   1:  PR[GP1:91,2] = PR[GP1:90,2] + -23.131;
   1:L PR[91] 10mm/sec CNT100;
   1:  PR[GP1:91,1] = PR[GP1:90,1] + -1.490;
   1:  PR[GP1:91,2] = PR[GP1:90,2] + -22.735;
   1:L PR[91] 10mm/sec CNT100;
   1:  PR[GP1:91,1] = PR[GP1:90,1] + 0.863;
   1:  PR[GP1:91,2] = PR[GP1:90,2] + -21.488;
   1:L PR[91] 10mm/sec CNT100;
   1:  PR[GP1:91,1] = PR[GP1:90,1] + 4.214;
   1:  PR[GP1:91,2] = PR[GP1:90,2] + -23.194;
   1:L PR[91] 10mm/sec CNT100;
   1:  PR[GP1:91,1] = PR[GP1:90,1] + 6.727;
   1:  PR[GP1:91,2] = PR[GP1:90,2] + -26.111;
   1:L PR[91] 10mm/sec CNT100;
   1:  PR[GP1:91,1] = PR[GP1:90,1] + 10.077;
   1:  PR[GP1:91,2] = PR[GP1:90,2] + -28.732;
   1:L PR[91] 10mm/sec CNT100;
   1:  PR[GP1:91,1] = PR[GP1:90,1] + 11.446;
   1:  PR[GP1:91,2] = PR[GP1:90,2] + -29.727;
   1:L PR[91] 10mm/sec CNT100;
   1:  PR[GP1:91,1] = PR[GP1:90,1] + 16.570;
   1:  PR[GP1:91,2] = PR[GP1:90,2] + -32.401;
   1:L PR[91] 10mm/sec CNT100;
   1:  PR[GP1:91,1] = PR[GP1:90,1] + 22.895;
   1:  PR[GP1:91,2] = PR[GP1:90,2] + -34.433;
   1:L PR[91] 10mm/sec CNT100;
   1:  PR[GP1:91,1] = PR[GP1:90,1] + 23.903;
   1:  PR[GP1:91,2] = PR[GP1:90,2] + -34.782;
   1:L PR[91] 10mm/sec CNT100;
   1:  PR[GP1:91,1] = PR[GP1:90,1] + 30.511;
   1:  PR[GP1:91,2] = PR[GP1:90,2] + -35.650;
   1:L PR[91] 10mm/sec CNT100;
   1:  PR[GP1:91,1] = PR[GP1:90,1] + 37.251;
   1:  PR[GP1:91,2] = PR[GP1:90,2] + -35.453;
   1:L PR[91] 10mm/sec CNT100;
   1:  PR[GP1:91,1] = PR[GP1:90,1] + 39.091;
   1:  PR[GP1:91,2] = PR[GP1:90,2] + -35.024;
   1:L PR[91] 10mm/sec CNT100;
   1:  PR[GP1:91,1] = PR[GP1:90,1] + 45.087;
   1:  PR[GP1:91,2] = PR[GP1:90,2] + -33.728;
   1:L PR[91] 10mm/sec CNT100;
   1:  PR[GP1:91,1] = PR[GP1:90,1] + 48.963;
   1:  PR[GP1:91,2] = PR[GP1:90,2] + -32.210;
   1:L PR[91] 10mm/sec CNT100;
   1:  PR[GP1:91,1] = PR[GP1:90,1] + 53.686;
   1:  PR[GP1:91,2] = PR[GP1:90,2] + -29.527;
   1:L PR[91] 10mm/sec CNT100;
   1:  PR[GP1:91,1] = PR[GP1:90,1] + 56.440;
   1:  PR[GP1:91,2] = PR[GP1:90,2] + -27.829;
   1:L PR[91] 10mm/sec CNT100;
   1:  PR[GP1:91,1] = PR[GP1:90,1] + 58.226;
   1:  PR[GP1:91,2] = PR[GP1:90,2] + -26.233;
   1:L PR[91] 10mm/sec CNT100;
   1:  PR[GP1:91,1] = PR[GP1:90,1] + 63.305;
   1:  PR[GP1:91,2] = PR[GP1:90,2] + -20.876;
   1:L PR[91] 10mm/sec CNT100;
   1:  PR[GP1:91,1] = PR[GP1:90,1] + 64.349;
   1:  PR[GP1:91,2] = PR[GP1:90,2] + -19.525;
   1:L PR[91] 10mm/sec CNT100;
   1:  PR[GP1:91,1] = PR[GP1:90,1] + 68.774;
   1:  PR[GP1:91,2] = PR[GP1:90,2] + -10.736;
   1:L PR[91] 10mm/sec CNT100;
   1:  PR[GP1:91,1] = PR[GP1:90,1] + 69.043;
   1:  PR[GP1:91,2] = PR[GP1:90,2] + -9.836;
   1:L PR[91] 10mm/sec CNT100;
   1:  PR[GP1:91,1] = PR[GP1:90,1] + 70.464;
   1:  PR[GP1:91,2] = PR[GP1:90,2] + -0.697;
   1:L PR[91] 10mm/sec CNT100;
   1:  PR[GP1:91,1] = PR[GP1:90,1] + 70.526;
   1:  PR[GP1:91,2] = PR[GP1:90,2] + -0.024;
   1:L PR[91] 10mm/sec CNT100;
   1:  PR[GP1:91,1] = PR[GP1:90,1] + 69.127;
   1:  PR[GP1:91,2] = PR[GP1:90,2] + 8.859;
   1:L PR[91] 10mm/sec CNT100;
   1:  PR[GP1:91,1] = PR[GP1:90,1] + 69.037;
   1:  PR[GP1:91,2] = PR[GP1:90,2] + 9.845;
   1:L PR[91] 10mm/sec CNT100;
   1:  PR[GP1:91,1] = PR[GP1:90,1] + 68.774;
   1:  PR[GP1:91,2] = PR[GP1:90,2] + 10.728;
   1:L PR[91] 10mm/sec CNT100;
   1:  PR[GP1:91,1] = PR[GP1:90,1] + 64.349;
   1:  PR[GP1:91,2] = PR[GP1:90,2] + 19.516;
   1:L PR[91] 10mm/sec CNT100;
   1:  PR[GP1:91,1] = PR[GP1:90,1] + 63.305;
   1:  PR[GP1:91,2] = PR[GP1:90,2] + 20.868;
   1:L PR[91] 10mm/sec CNT100;
   1:  PR[GP1:91,1] = PR[GP1:90,1] + 58.226;
   1:  PR[GP1:91,2] = PR[GP1:90,2] + 26.224;
   1:L PR[91] 10mm/sec CNT100;
   1:  PR[GP1:91,1] = PR[GP1:90,1] + 56.449;
   1:  PR[GP1:91,2] = PR[GP1:90,2] + 27.812;
   1:L PR[91] 10mm/sec CNT100;
   1:  PR[GP1:91,1] = PR[GP1:90,1] + 51.595;
   1:  PR[GP1:91,2] = PR[GP1:90,2] + 30.539;
   1:L PR[91] 10mm/sec CNT100;
   1:  PR[GP1:91,1] = PR[GP1:90,1] + 48.950;
   1:  PR[GP1:91,2] = PR[GP1:90,2] + 32.206;
   1:L PR[91] 10mm/sec CNT100;
   1:  PR[GP1:91,1] = PR[GP1:90,1] + 45.081;
   1:  PR[GP1:91,2] = PR[GP1:90,2] + 33.721;
   1:L PR[91] 10mm/sec CNT100;
   1:  PR[GP1:91,1] = PR[GP1:90,1] + 41.998;
   1:  PR[GP1:91,2] = PR[GP1:90,2] + 34.448;
   1:L PR[91] 10mm/sec CNT100;
   1:  PR[GP1:91,1] = PR[GP1:90,1] + 37.257;
   1:  PR[GP1:91,2] = PR[GP1:90,2] + 35.444;
   1:L PR[91] 10mm/sec CNT100;
   1:  PR[GP1:91,1] = PR[GP1:90,1] + 30.511;
   1:  PR[GP1:91,2] = PR[GP1:90,2] + 35.642;
   1:L PR[91] 10mm/sec CNT100;
   1:  PR[GP1:91,1] = PR[GP1:90,1] + 23.897;
   1:  PR[GP1:91,2] = PR[GP1:90,2] + 34.772;
   1:L PR[91] 10mm/sec CNT100;
   1:  PR[GP1:91,1] = PR[GP1:90,1] + 18.223;
   1:  PR[GP1:91,2] = PR[GP1:90,2] + 32.967;
   1:L PR[91] 10mm/sec CNT100;
   1:  PR[GP1:91,1] = PR[GP1:90,1] + 16.579;
   1:  PR[GP1:91,2] = PR[GP1:90,2] + 32.397;
   1:L PR[91] 10mm/sec CNT100;
   1:  PR[GP1:91,1] = PR[GP1:90,1] + 11.445;
   1:  PR[GP1:91,2] = PR[GP1:90,2] + 29.717;
   1:L PR[91] 10mm/sec CNT100;
   1:  PR[GP1:91,1] = PR[GP1:90,1] + 10.460;
   1:  PR[GP1:91,2] = PR[GP1:90,2] + 29.022;
   1:L PR[91] 10mm/sec CNT100;
   1:  PR[GP1:91,1] = PR[GP1:90,1] + 6.917;
   1:  PR[GP1:91,2] = PR[GP1:90,2] + 26.249;
   1:L PR[91] 10mm/sec CNT100;
   1:  PR[GP1:91,1] = PR[GP1:90,1] + 4.197;
   1:  PR[GP1:91,2] = PR[GP1:90,2] + 23.083;
   1:L PR[91] 10mm/sec CNT100;
   1:  PR[GP1:91,1] = PR[GP1:90,1] + 3.346;
   1:  PR[GP1:91,2] = PR[GP1:90,2] + 22.747;
   1:L PR[91] 10mm/sec CNT100;
   1:  PR[GP1:91,1] = PR[GP1:90,1] + 0.976;
   1:  PR[GP1:91,2] = PR[GP1:90,2] + 21.536;
   1:L PR[91] 10mm/sec CNT100;
   1:  PR[GP1:91,1] = PR[GP1:90,1] + -0.928;
   1:  PR[GP1:91,2] = PR[GP1:90,2] + 22.512;
   1:  PR[GP1:91,3] = PR[GP1:90,3] + 46.550;
   1:L PR[91] 10mm/sec CNT100;
   1:  PR[GP1:91,1] = PR[GP1:90,1] + -3.325;
   1:  PR[GP1:91,2] = PR[GP1:90,2] + 23.731;
   1:L PR[91] 10mm/sec CNT100;
   1:  PR[GP1:91,1] = PR[GP1:90,1] + -5.725;
   1:  PR[GP1:91,2] = PR[GP1:90,2] + 26.522;
   1:L PR[91] 10mm/sec CNT100;
   1:  PR[GP1:91,1] = PR[GP1:90,1] + -8.906;
   1:  PR[GP1:91,2] = PR[GP1:90,2] + 29.013;
   1:L PR[91] 10mm/sec CNT100;
   1:  PR[GP1:91,1] = PR[GP1:90,1] + -10.149;
   1:  PR[GP1:91,2] = PR[GP1:90,2] + 29.891;
   1:L PR[91] 10mm/sec CNT100;
   1:  PR[GP1:91,1] = PR[GP1:90,1] + -15.022;
   1:  PR[GP1:91,2] = PR[GP1:90,2] + 32.441;
   1:L PR[91] 10mm/sec CNT100;
   1:  PR[GP1:91,1] = PR[GP1:90,1] + -20.991;
   1:  PR[GP1:91,2] = PR[GP1:90,2] + 34.359;
   1:L PR[91] 10mm/sec CNT100;
   1:  PR[GP1:91,1] = PR[GP1:90,1] + -22.656;
   1:  PR[GP1:91,2] = PR[GP1:90,2] + 34.934;
   1:L PR[91] 10mm/sec CNT100;
   1:  PR[GP1:91,1] = PR[GP1:90,1] + -28.937;
   1:  PR[GP1:91,2] = PR[GP1:90,2] + 35.755;
   1:L PR[91] 10mm/sec CNT100;
   1:  PR[GP1:91,1] = PR[GP1:90,1] + -36.208;
   1:  PR[GP1:91,2] = PR[GP1:90,2] + 35.505;
   1:L PR[91] 10mm/sec CNT100;
   1:  PR[GP1:91,1] = PR[GP1:90,1] + -43.441;
   1:  PR[GP1:91,2] = PR[GP1:90,2] + 33.938;
   1:L PR[91] 10mm/sec CNT100;
   1:  PR[GP1:91,1] = PR[GP1:90,1] + -48.169;
   1:  PR[GP1:91,2] = PR[GP1:90,2] + 32.077;
   1:L PR[91] 10mm/sec CNT100;
   1:  PR[GP1:91,1] = PR[GP1:90,1] + -51.524;
   1:  PR[GP1:91,2] = PR[GP1:90,2] + 30.168;
   1:L PR[91] 10mm/sec CNT100;
   1:  PR[GP1:91,1] = PR[GP1:90,1] + -55.181;
   1:  PR[GP1:91,2] = PR[GP1:90,2] + 27.903;
   1:L PR[91] 10mm/sec CNT100;
   1:  PR[GP1:91,1] = PR[GP1:90,1] + -57.555;
   1:  PR[GP1:91,2] = PR[GP1:90,2] + 25.775;
   1:L PR[91] 10mm/sec CNT100;
   1:  PR[GP1:91,1] = PR[GP1:90,1] + -61.710;
   1:  PR[GP1:91,2] = PR[GP1:90,2] + 21.407;
   1:L PR[91] 10mm/sec CNT100;
   1:  PR[GP1:91,1] = PR[GP1:90,1] + -63.266;
   1:  PR[GP1:91,2] = PR[GP1:90,2] + 19.387;
   1:L PR[91] 10mm/sec CNT100;
   1:  PR[GP1:91,1] = PR[GP1:90,1] + -67.485;
   1:  PR[GP1:91,2] = PR[GP1:90,2] + 10.965;
   1:L PR[91] 10mm/sec CNT100;
   1:  PR[GP1:91,1] = PR[GP1:90,1] + -67.973;
   1:  PR[GP1:91,2] = PR[GP1:90,2] + 9.309;
   1:L PR[91] 10mm/sec CNT100;
   1:  PR[GP1:91,1] = PR[GP1:90,1] + -69.196;
   1:  PR[GP1:91,2] = PR[GP1:90,2] + 1.460;
   1:L PR[91] 10mm/sec CNT100;
   1:  PR[GP1:91,1] = PR[GP1:90,1] + -69.326;
   1:  PR[GP1:91,2] = PR[GP1:90,2] + 0.016;
   1:L PR[91] 10mm/sec CNT100;
   1:  PR[GP1:91,1] = PR[GP1:90,1] + -68.117;
   1:  PR[GP1:91,2] = PR[GP1:90,2] + -7.637;
   1:L PR[91] 10mm/sec CNT100;
   1:  PR[GP1:91,1] = PR[GP1:90,1] + -67.967;
   1:  PR[GP1:91,2] = PR[GP1:90,2] + -9.337;
   1:L PR[91] 10mm/sec CNT100;
   1:  PR[GP1:91,1] = PR[GP1:90,1] + -67.485;
   1:  PR[GP1:91,2] = PR[GP1:90,2] + -10.974;
   1:L PR[91] 10mm/sec CNT100;
   1:  PR[GP1:91,1] = PR[GP1:90,1] + -63.266;
   1:  PR[GP1:91,2] = PR[GP1:90,2] + -19.396;
   1:L PR[91] 10mm/sec CNT100;
   1:  PR[GP1:91,1] = PR[GP1:90,1] + -61.710;
   1:  PR[GP1:91,2] = PR[GP1:90,2] + -21.416;
   1:L PR[91] 10mm/sec CNT100;
   1:  PR[GP1:91,1] = PR[GP1:90,1] + -57.555;
   1:  PR[GP1:91,2] = PR[GP1:90,2] + -25.784;
   1:L PR[91] 10mm/sec CNT100;
   1:  PR[GP1:91,1] = PR[GP1:90,1] + -55.191;
   1:  PR[GP1:91,2] = PR[GP1:90,2] + -27.903;
   1:L PR[91] 10mm/sec CNT100;
   1:  PR[GP1:91,1] = PR[GP1:90,1] + -51.401;
   1:  PR[GP1:91,2] = PR[GP1:90,2] + -30.035;
   1:L PR[91] 10mm/sec CNT100;
   1:  PR[GP1:91,1] = PR[GP1:90,1] + -48.156;
   1:  PR[GP1:91,2] = PR[GP1:90,2] + -32.091;
   1:L PR[91] 10mm/sec CNT100;
   1:  PR[GP1:91,1] = PR[GP1:90,1] + -43.436;
   1:  PR[GP1:91,2] = PR[GP1:90,2] + -33.949;
   1:L PR[91] 10mm/sec CNT100;
   1:  PR[GP1:91,1] = PR[GP1:90,1] + -41.730;
   1:  PR[GP1:91,2] = PR[GP1:90,2] + -34.350;
   1:L PR[91] 10mm/sec CNT100;
   1:  PR[GP1:91,1] = PR[GP1:90,1] + -36.208;
   1:  PR[GP1:91,2] = PR[GP1:90,2] + -35.514;
   1:L PR[91] 10mm/sec CNT100;
   1:  PR[GP1:91,1] = PR[GP1:90,1] + -29.774;
   1:  PR[GP1:91,2] = PR[GP1:90,2] + -35.762;
   1:L PR[91] 10mm/sec CNT100;
   1:  PR[GP1:91,1] = PR[GP1:90,1] + -28.945;
   1:  PR[GP1:91,2] = PR[GP1:90,2] + -35.765;
   1:L PR[91] 10mm/sec CNT100;
   1:  PR[GP1:91,1] = PR[GP1:90,1] + -22.646;
   1:  PR[GP1:91,2] = PR[GP1:90,2] + -34.942;
   1:L PR[91] 10mm/sec CNT100;
   1:  PR[GP1:91,1] = PR[GP1:90,1] + -17.264;
   1:  PR[GP1:91,2] = PR[GP1:90,2] + -33.229;
   1:L PR[91] 10mm/sec CNT100;
   1:  PR[GP1:91,1] = PR[GP1:90,1] + -15.025;
   1:  PR[GP1:91,2] = PR[GP1:90,2] + -32.451;
   1:L PR[91] 10mm/sec CNT100;
   1:  PR[GP1:91,1] = PR[GP1:90,1] + -10.150;
   1:  PR[GP1:91,2] = PR[GP1:90,2] + -29.900;
   1:L PR[91] 10mm/sec CNT100;
   1:  PR[GP1:91,1] = PR[GP1:90,1] + -8.426;
   1:  PR[GP1:91,2] = PR[GP1:90,2] + -28.648;
   1:L PR[91] 10mm/sec CNT100;
   1:  PR[GP1:91,1] = PR[GP1:90,1] + -5.499;
   1:  PR[GP1:91,2] = PR[GP1:90,2] + -26.355;
   1:L PR[91] 10mm/sec CNT100;
   1:  PR[GP1:91,1] = PR[GP1:90,1] + -3.269;
   1:  PR[GP1:91,2] = PR[GP1:90,2] + -23.769;
   1:L PR[91] 10mm/sec CNT100;
   1:  PR[GP1:91,1] = PR[GP1:90,1] + -1.127;
   1:  PR[GP1:91,2] = PR[GP1:90,2] + -23.309;
   1:L PR[91] 10mm/sec CNT100;
   1:  PR[GP1:91,1] = PR[GP1:90,1] + 0.953;
   1:  PR[GP1:91,2] = PR[GP1:90,2] + -22.208;
   1:L PR[91] 10mm/sec CNT100;
   1:  PR[GP1:91,1] = PR[GP1:90,1] + 4.149;
   1:  PR[GP1:91,2] = PR[GP1:90,2] + -23.833;
   1:L PR[91] 10mm/sec CNT100;
   1:  PR[GP1:91,1] = PR[GP1:90,1] + 6.345;
   1:  PR[GP1:91,2] = PR[GP1:90,2] + -26.382;
   1:L PR[91] 10mm/sec CNT100;
   1:  PR[GP1:91,1] = PR[GP1:90,1] + 9.258;
   1:  PR[GP1:91,2] = PR[GP1:90,2] + -28.661;
   1:L PR[91] 10mm/sec CNT100;
   1:  PR[GP1:91,1] = PR[GP1:90,1] + 10.985;
   1:  PR[GP1:91,2] = PR[GP1:90,2] + -29.916;
   1:L PR[91] 10mm/sec CNT100;
   1:  PR[GP1:91,1] = PR[GP1:90,1] + 15.824;
   1:  PR[GP1:91,2] = PR[GP1:90,2] + -32.441;
   1:L PR[91] 10mm/sec CNT100;
   1:  PR[GP1:91,1] = PR[GP1:90,1] + 21.801;
   1:  PR[GP1:91,2] = PR[GP1:90,2] + -34.362;
   1:L PR[91] 10mm/sec CNT100;
   1:  PR[GP1:91,1] = PR[GP1:90,1] + 23.469;
   1:  PR[GP1:91,2] = PR[GP1:90,2] + -34.939;
   1:L PR[91] 10mm/sec CNT100;
   1:  PR[GP1:91,1] = PR[GP1:90,1] + 29.742;
   1:  PR[GP1:91,2] = PR[GP1:90,2] + -35.764;
   1:L PR[91] 10mm/sec CNT100;
   1:  PR[GP1:91,1] = PR[GP1:90,1] + 36.985;
   1:  PR[GP1:91,2] = PR[GP1:90,2] + -35.521;
   1:L PR[91] 10mm/sec CNT100;
   1:  PR[GP1:91,1] = PR[GP1:90,1] + 44.219;
   1:  PR[GP1:91,2] = PR[GP1:90,2] + -33.956;
   1:L PR[91] 10mm/sec CNT100;
   1:  PR[GP1:91,1] = PR[GP1:90,1] + 48.968;
   1:  PR[GP1:91,2] = PR[GP1:90,2] + -32.097;
   1:L PR[91] 10mm/sec CNT100;
   1:  PR[GP1:91,1] = PR[GP1:90,1] + 52.319;
   1:  PR[GP1:91,2] = PR[GP1:90,2] + -30.193;
   1:L PR[91] 10mm/sec CNT100;
   1:  PR[GP1:91,1] = PR[GP1:90,1] + 55.967;
   1:  PR[GP1:91,2] = PR[GP1:90,2] + -27.944;
   1:L PR[91] 10mm/sec CNT100;
   1:  PR[GP1:91,1] = PR[GP1:90,1] + 58.339;
   1:  PR[GP1:91,2] = PR[GP1:90,2] + -25.825;
   1:L PR[91] 10mm/sec CNT100;
   1:  PR[GP1:91,1] = PR[GP1:90,1] + 62.493;
   1:  PR[GP1:91,2] = PR[GP1:90,2] + -21.443;
   1:L PR[91] 10mm/sec CNT100;
   1:  PR[GP1:91,1] = PR[GP1:90,1] + 64.073;
   1:  PR[GP1:91,2] = PR[GP1:90,2] + -19.399;
   1:L PR[91] 10mm/sec CNT100;
   1:  PR[GP1:91,1] = PR[GP1:90,1] + 67.337;
   1:  PR[GP1:91,2] = PR[GP1:90,2] + -12.902;
   1:L PR[91] 10mm/sec CNT100;
   1:  PR[GP1:91,1] = PR[GP1:90,1] + 68.299;
   1:  PR[GP1:91,2] = PR[GP1:90,2] + -11.018;
   1:L PR[91] 10mm/sec CNT100;
   1:  PR[GP1:91,1] = PR[GP1:90,1] + 68.786;
   1:  PR[GP1:91,2] = PR[GP1:90,2] + -9.386;
   1:L PR[91] 10mm/sec CNT100;
   1:  PR[GP1:91,1] = PR[GP1:90,1] + 70.010;
   1:  PR[GP1:91,2] = PR[GP1:90,2] + -1.512;
   1:L PR[91] 10mm/sec CNT100;
   1:  PR[GP1:91,1] = PR[GP1:90,1] + 70.147;
   1:  PR[GP1:91,2] = PR[GP1:90,2] + -0.024;
   1:L PR[91] 10mm/sec CNT100;
   1:  PR[GP1:91,1] = PR[GP1:90,1] + 68.938;
   1:  PR[GP1:91,2] = PR[GP1:90,2] + 7.649;
   1:L PR[91] 10mm/sec CNT100;
   1:  PR[GP1:91,1] = PR[GP1:90,1] + 68.780;
   1:  PR[GP1:91,2] = PR[GP1:90,2] + 9.396;
   1:L PR[91] 10mm/sec CNT100;
   1:  PR[GP1:91,1] = PR[GP1:90,1] + 68.298;
   1:  PR[GP1:91,2] = PR[GP1:90,2] + 11.011;
   1:L PR[91] 10mm/sec CNT100;
   1:  PR[GP1:91,1] = PR[GP1:90,1] + 65.100;
   1:  PR[GP1:91,2] = PR[GP1:90,2] + 17.382;
   1:L PR[91] 10mm/sec CNT100;
   1:  PR[GP1:91,1] = PR[GP1:90,1] + 64.074;
   1:  PR[GP1:91,2] = PR[GP1:90,2] + 19.388;
   1:L PR[91] 10mm/sec CNT100;
   1:  PR[GP1:91,1] = PR[GP1:90,1] + 62.493;
   1:  PR[GP1:91,2] = PR[GP1:90,2] + 21.434;
   1:L PR[91] 10mm/sec CNT100;
   1:  PR[GP1:91,1] = PR[GP1:90,1] + 58.339;
   1:  PR[GP1:91,2] = PR[GP1:90,2] + 25.816;
   1:L PR[91] 10mm/sec CNT100;
   1:  PR[GP1:91,1] = PR[GP1:90,1] + 55.976;
   1:  PR[GP1:91,2] = PR[GP1:90,2] + 27.927;
   1:L PR[91] 10mm/sec CNT100;
   1:  PR[GP1:91,1] = PR[GP1:90,1] + 52.190;
   1:  PR[GP1:91,2] = PR[GP1:90,2] + 30.054;
   1:L PR[91] 10mm/sec CNT100;
   1:  PR[GP1:91,1] = PR[GP1:90,1] + 48.955;
   1:  PR[GP1:91,2] = PR[GP1:90,2] + 32.093;
   1:L PR[91] 10mm/sec CNT100;
   1:  PR[GP1:91,1] = PR[GP1:90,1] + 44.214;
   1:  PR[GP1:91,2] = PR[GP1:90,2] + 33.949;
   1:L PR[91] 10mm/sec CNT100;
   1:  PR[GP1:91,1] = PR[GP1:90,1] + 42.517;
   1:  PR[GP1:91,2] = PR[GP1:90,2] + 34.349;
   1:L PR[91] 10mm/sec CNT100;
   1:  PR[GP1:91,1] = PR[GP1:90,1] + 36.985;
   1:  PR[GP1:91,2] = PR[GP1:90,2] + 35.512;
   1:L PR[91] 10mm/sec CNT100;
   1:  PR[GP1:91,1] = PR[GP1:90,1] + 30.583;
   1:  PR[GP1:91,2] = PR[GP1:90,2] + 35.753;
   1:L PR[91] 10mm/sec CNT100;
   1:  PR[GP1:91,1] = PR[GP1:90,1] + 29.753;
   1:  PR[GP1:91,2] = PR[GP1:90,2] + 35.756;
   1:L PR[91] 10mm/sec CNT100;
   1:  PR[GP1:91,1] = PR[GP1:90,1] + 23.464;
   1:  PR[GP1:91,2] = PR[GP1:90,2] + 34.930;
   1:L PR[91] 10mm/sec CNT100;
   1:  PR[GP1:91,1] = PR[GP1:90,1] + 18.075;
   1:  PR[GP1:91,2] = PR[GP1:90,2] + 33.215;
   1:L PR[91] 10mm/sec CNT100;
   1:  PR[GP1:91,1] = PR[GP1:90,1] + 15.834;
   1:  PR[GP1:91,2] = PR[GP1:90,2] + 32.438;
   1:L PR[91] 10mm/sec CNT100;
   1:  PR[GP1:91,1] = PR[GP1:90,1] + 10.984;
   1:  PR[GP1:91,2] = PR[GP1:90,2] + 29.907;
   1:L PR[91] 10mm/sec CNT100;
   1:  PR[GP1:91,1] = PR[GP1:90,1] + 9.739;
   1:  PR[GP1:91,2] = PR[GP1:90,2] + 29.027;
   1:L PR[91] 10mm/sec CNT100;
   1:  PR[GP1:91,1] = PR[GP1:90,1] + 6.573;
   1:  PR[GP1:91,2] = PR[GP1:90,2] + 26.550;
   1:L PR[91] 10mm/sec CNT100;
   1:  PR[GP1:91,1] = PR[GP1:90,1] + 4.132;
   1:  PR[GP1:91,2] = PR[GP1:90,2] + 23.708;
   1:L PR[91] 10mm/sec CNT100;
   1:  PR[GP1:91,1] = PR[GP1:90,1] + 3.152;
   1:  PR[GP1:91,2] = PR[GP1:90,2] + 23.322;
   1:L PR[91] 10mm/sec CNT100;
   1:  PR[GP1:91,1] = PR[GP1:90,1] + 1.066;
   1:  PR[GP1:91,2] = PR[GP1:90,2] + 22.256;
   1:L PR[91] 10mm/sec CNT100;
   1:  PR[GP1:91,1] = PR[GP1:90,1] + -1.121;
   1:  PR[GP1:91,2] = PR[GP1:90,2] + 23.268;
   1:  PR[GP1:91,3] = PR[GP1:90,3] + 47.880;
   1:L PR[91] 10mm/sec CNT100;
   1:  PR[GP1:91,1] = PR[GP1:90,1] + -3.261;
   1:  PR[GP1:91,2] = PR[GP1:90,2] + 24.356;
   1:L PR[91] 10mm/sec CNT100;
   1:  PR[GP1:91,1] = PR[GP1:90,1] + -5.385;
   1:  PR[GP1:91,2] = PR[GP1:90,2] + 26.826;
   1:L PR[91] 10mm/sec CNT100;
   1:  PR[GP1:91,1] = PR[GP1:90,1] + -8.188;
   1:  PR[GP1:91,2] = PR[GP1:90,2] + 29.021;
   1:L PR[91] 10mm/sec CNT100;
   1:  PR[GP1:91,1] = PR[GP1:90,1] + -9.689;
   1:  PR[GP1:91,2] = PR[GP1:90,2] + 30.082;
   1:L PR[91] 10mm/sec CNT100;
   1:  PR[GP1:91,1] = PR[GP1:90,1] + -14.277;
   1:  PR[GP1:91,2] = PR[GP1:90,2] + 32.482;
   1:L PR[91] 10mm/sec CNT100;
   1:  PR[GP1:91,1] = PR[GP1:90,1] + -19.899;
   1:  PR[GP1:91,2] = PR[GP1:90,2] + 34.288;
   1:L PR[91] 10mm/sec CNT100;
   1:  PR[GP1:91,1] = PR[GP1:90,1] + -22.224;
   1:  PR[GP1:91,2] = PR[GP1:90,2] + 35.092;
   1:L PR[91] 10mm/sec CNT100;
   1:  PR[GP1:91,1] = PR[GP1:90,1] + -28.171;
   1:  PR[GP1:91,2] = PR[GP1:90,2] + 35.869;
   1:L PR[91] 10mm/sec CNT100;
   1:  PR[GP1:91,1] = PR[GP1:90,1] + -35.111;
   1:  PR[GP1:91,2] = PR[GP1:90,2] + 35.630;
   1:L PR[91] 10mm/sec CNT100;
   1:  PR[GP1:91,1] = PR[GP1:90,1] + -35.807;
   1:  PR[GP1:91,2] = PR[GP1:90,2] + 35.627;
   1:L PR[91] 10mm/sec CNT100;
   1:  PR[GP1:91,1] = PR[GP1:90,1] + -42.581;
   1:  PR[GP1:91,2] = PR[GP1:90,2] + 34.164;
   1:L PR[91] 10mm/sec CNT100;
   1:  PR[GP1:91,1] = PR[GP1:90,1] + -48.178;
   1:  PR[GP1:91,2] = PR[GP1:90,2] + 31.961;
   1:L PR[91] 10mm/sec CNT100;
   1:  PR[GP1:91,1] = PR[GP1:90,1] + -50.163;
   1:  PR[GP1:91,2] = PR[GP1:90,2] + 30.832;
   1:L PR[91] 10mm/sec CNT100;
   1:  PR[GP1:91,1] = PR[GP1:90,1] + -54.716;
   1:  PR[GP1:91,2] = PR[GP1:90,2] + 28.012;
   1:L PR[91] 10mm/sec CNT100;
   1:  PR[GP1:91,1] = PR[GP1:90,1] + -57.676;
   1:  PR[GP1:91,2] = PR[GP1:90,2] + 25.358;
   1:L PR[91] 10mm/sec CNT100;
   1:  PR[GP1:91,1] = PR[GP1:90,1] + -60.910;
   1:  PR[GP1:91,2] = PR[GP1:90,2] + 21.959;
   1:L PR[91] 10mm/sec CNT100;
   1:  PR[GP1:91,1] = PR[GP1:90,1] + -62.994;
   1:  PR[GP1:91,2] = PR[GP1:90,2] + 19.254;
   1:L PR[91] 10mm/sec CNT100;
   1:  PR[GP1:91,1] = PR[GP1:90,1] + -67.013;
   1:  PR[GP1:91,2] = PR[GP1:90,2] + 11.241;
   1:L PR[91] 10mm/sec CNT100;
   1:  PR[GP1:91,1] = PR[GP1:90,1] + -67.719;
   1:  PR[GP1:91,2] = PR[GP1:90,2] + 8.842;
   1:L PR[91] 10mm/sec CNT100;
   1:  PR[GP1:91,1] = PR[GP1:90,1] + -68.746;
   1:  PR[GP1:91,2] = PR[GP1:90,2] + 2.253;
   1:L PR[91] 10mm/sec CNT100;
   1:  PR[GP1:91,1] = PR[GP1:90,1] + -68.947;
   1:  PR[GP1:91,2] = PR[GP1:90,2] + 0.016;
   1:L PR[91] 10mm/sec CNT100;
   1:  PR[GP1:91,1] = PR[GP1:90,1] + -67.929;
   1:  PR[GP1:91,2] = PR[GP1:90,2] + -6.431;
   1:L PR[91] 10mm/sec CNT100;
   1:  PR[GP1:91,1] = PR[GP1:90,1] + -67.713;
   1:  PR[GP1:91,2] = PR[GP1:90,2] + -8.870;
   1:L PR[91] 10mm/sec CNT100;
   1:  PR[GP1:91,1] = PR[GP1:90,1] + -67.013;
   1:  PR[GP1:91,2] = PR[GP1:90,2] + -11.249;
   1:L PR[91] 10mm/sec CNT100;
   1:  PR[GP1:91,1] = PR[GP1:90,1] + -62.994;
   1:  PR[GP1:91,2] = PR[GP1:90,2] + -19.262;
   1:L PR[91] 10mm/sec CNT100;
   1:  PR[GP1:91,1] = PR[GP1:90,1] + -60.910;
   1:  PR[GP1:91,2] = PR[GP1:90,2] + -21.968;
   1:L PR[91] 10mm/sec CNT100;
   1:  PR[GP1:91,1] = PR[GP1:90,1] + -57.676;
   1:  PR[GP1:91,2] = PR[GP1:90,2] + -25.367;
   1:L PR[91] 10mm/sec CNT100;
   1:  PR[GP1:91,1] = PR[GP1:90,1] + -54.726;
   1:  PR[GP1:91,2] = PR[GP1:90,2] + -28.012;
   1:L PR[91] 10mm/sec CNT100;
   1:  PR[GP1:91,1] = PR[GP1:90,1] + -52.003;
   1:  PR[GP1:91,2] = PR[GP1:90,2] + -29.544;
   1:L PR[91] 10mm/sec CNT100;
   1:  PR[GP1:91,1] = PR[GP1:90,1] + -48.165;
   1:  PR[GP1:91,2] = PR[GP1:90,2] + -31.975;
   1:L PR[91] 10mm/sec CNT100;
   1:  PR[GP1:91,1] = PR[GP1:90,1] + -42.581;
   1:  PR[GP1:91,2] = PR[GP1:90,2] + -34.173;
   1:L PR[91] 10mm/sec CNT100;
   1:  PR[GP1:91,1] = PR[GP1:90,1] + -35.796;
   1:  PR[GP1:91,2] = PR[GP1:90,2] + -35.638;
   1:L PR[91] 10mm/sec CNT100;
   1:  PR[GP1:91,1] = PR[GP1:90,1] + -29.674;
   1:  PR[GP1:91,2] = PR[GP1:90,2] + -35.874;
   1:L PR[91] 10mm/sec CNT100;
   1:  PR[GP1:91,1] = PR[GP1:90,1] + -28.177;
   1:  PR[GP1:91,2] = PR[GP1:90,2] + -35.879;
   1:L PR[91] 10mm/sec CNT100;
   1:  PR[GP1:91,1] = PR[GP1:90,1] + -22.212;
   1:  PR[GP1:91,2] = PR[GP1:90,2] + -35.099;
   1:L PR[91] 10mm/sec CNT100;
   1:  PR[GP1:91,1] = PR[GP1:90,1] + -17.114;
   1:  PR[GP1:91,2] = PR[GP1:90,2] + -33.477;
   1:L PR[91] 10mm/sec CNT100;
   1:  PR[GP1:91,1] = PR[GP1:90,1] + -14.279;
   1:  PR[GP1:91,2] = PR[GP1:90,2] + -32.491;
   1:L PR[91] 10mm/sec CNT100;
   1:  PR[GP1:91,1] = PR[GP1:90,1] + -9.690;
   1:  PR[GP1:91,2] = PR[GP1:90,2] + -30.090;
   1:L PR[91] 10mm/sec CNT100;
   1:  PR[GP1:91,1] = PR[GP1:90,1] + -7.610;
   1:  PR[GP1:91,2] = PR[GP1:90,2] + -28.580;
   1:L PR[91] 10mm/sec CNT100;
   1:  PR[GP1:91,1] = PR[GP1:90,1] + -5.121;
   1:  PR[GP1:91,2] = PR[GP1:90,2] + -26.630;
   1:L PR[91] 10mm/sec CNT100;
   1:  PR[GP1:91,1] = PR[GP1:90,1] + -3.205;
   1:  PR[GP1:91,2] = PR[GP1:90,2] + -24.408;
   1:L PR[91] 10mm/sec CNT100;
   1:  PR[GP1:91,1] = PR[GP1:90,1] + -0.763;
   1:  PR[GP1:91,2] = PR[GP1:90,2] + -23.884;
   1:L PR[91] 10mm/sec CNT100;
   1:  PR[GP1:91,1] = PR[GP1:90,1] + 1.043;
   1:  PR[GP1:91,2] = PR[GP1:90,2] + -22.927;
   1:L PR[91] 10mm/sec CNT100;
   1:  PR[GP1:91,1] = PR[GP1:90,1] + 4.084;
   1:  PR[GP1:91,2] = PR[GP1:90,2] + -24.471;
   1:L PR[91] 10mm/sec CNT100;
   1:  PR[GP1:91,1] = PR[GP1:90,1] + 5.962;
   1:  PR[GP1:91,2] = PR[GP1:90,2] + -26.653;
   1:L PR[91] 10mm/sec CNT100;
   1:  PR[GP1:91,1] = PR[GP1:90,1] + 8.440;
   1:  PR[GP1:91,2] = PR[GP1:90,2] + -28.591;
   1:L PR[91] 10mm/sec CNT100;
   1:  PR[GP1:91,1] = PR[GP1:90,1] + 10.524;
   1:  PR[GP1:91,2] = PR[GP1:90,2] + -30.105;
   1:L PR[91] 10mm/sec CNT100;
   1:  PR[GP1:91,1] = PR[GP1:90,1] + 15.078;
   1:  PR[GP1:91,2] = PR[GP1:90,2] + -32.482;
   1:L PR[91] 10mm/sec CNT100;
   1:  PR[GP1:91,1] = PR[GP1:90,1] + 20.708;
   1:  PR[GP1:91,2] = PR[GP1:90,2] + -34.291;
   1:L PR[91] 10mm/sec CNT100;
   1:  PR[GP1:91,1] = PR[GP1:90,1] + 23.036;
   1:  PR[GP1:91,2] = PR[GP1:90,2] + -35.097;
   1:L PR[91] 10mm/sec CNT100;
   1:  PR[GP1:91,1] = PR[GP1:90,1] + 28.975;
   1:  PR[GP1:91,2] = PR[GP1:90,2] + -35.877;
   1:L PR[91] 10mm/sec CNT100;
   1:  PR[GP1:91,1] = PR[GP1:90,1] + 35.883;
   1:  PR[GP1:91,2] = PR[GP1:90,2] + -35.645;
   1:L PR[91] 10mm/sec CNT100;
   1:  PR[GP1:91,1] = PR[GP1:90,1] + 36.585;
   1:  PR[GP1:91,2] = PR[GP1:90,2] + -35.642;
   1:L PR[91] 10mm/sec CNT100;
   1:  PR[GP1:91,1] = PR[GP1:90,1] + 43.352;
   1:  PR[GP1:91,2] = PR[GP1:90,2] + -34.184;
   1:L PR[91] 10mm/sec CNT100;
   1:  PR[GP1:91,1] = PR[GP1:90,1] + 48.973;
   1:  PR[GP1:91,2] = PR[GP1:90,2] + -31.984;
   1:L PR[91] 10mm/sec CNT100;
   1:  PR[GP1:91,1] = PR[GP1:90,1] + 50.952;
   1:  PR[GP1:91,2] = PR[GP1:90,2] + -30.859;
   1:L PR[91] 10mm/sec CNT100;
   1:  PR[GP1:91,1] = PR[GP1:90,1] + 55.493;
   1:  PR[GP1:91,2] = PR[GP1:90,2] + -28.059;
   1:L PR[91] 10mm/sec CNT100;
   1:  PR[GP1:91,1] = PR[GP1:90,1] + 58.451;
   1:  PR[GP1:91,2] = PR[GP1:90,2] + -25.416;
   1:L PR[91] 10mm/sec CNT100;
   1:  PR[GP1:91,1] = PR[GP1:90,1] + 61.681;
   1:  PR[GP1:91,2] = PR[GP1:90,2] + -22.010;
   1:L PR[91] 10mm/sec CNT100;
   1:  PR[GP1:91,1] = PR[GP1:90,1] + 63.796;
   1:  PR[GP1:91,2] = PR[GP1:90,2] + -19.272;
   1:L PR[91] 10mm/sec CNT100;
   1:  PR[GP1:91,1] = PR[GP1:90,1] + 66.443;
   1:  PR[GP1:91,2] = PR[GP1:90,2] + -14.006;
   1:L PR[91] 10mm/sec CNT100;
   1:  PR[GP1:91,1] = PR[GP1:90,1] + 67.823;
   1:  PR[GP1:91,2] = PR[GP1:90,2] + -11.301;
   1:L PR[91] 10mm/sec CNT100;
   1:  PR[GP1:91,1] = PR[GP1:90,1] + 68.528;
   1:  PR[GP1:91,2] = PR[GP1:90,2] + -8.937;
   1:L PR[91] 10mm/sec CNT100;
   1:  PR[GP1:91,1] = PR[GP1:90,1] + 69.556;
   1:  PR[GP1:91,2] = PR[GP1:90,2] + -2.327;
   1:L PR[91] 10mm/sec CNT100;
   1:  PR[GP1:91,1] = PR[GP1:90,1] + 69.768;
   1:  PR[GP1:91,2] = PR[GP1:90,2] + -0.024;
   1:L PR[91] 10mm/sec CNT100;
   1:  PR[GP1:91,1] = PR[GP1:90,1] + 68.749;
   1:  PR[GP1:91,2] = PR[GP1:90,2] + 6.440;
   1:L PR[91] 10mm/sec CNT100;
   1:  PR[GP1:91,1] = PR[GP1:90,1] + 68.523;
   1:  PR[GP1:91,2] = PR[GP1:90,2] + 8.946;
   1:L PR[91] 10mm/sec CNT100;
   1:  PR[GP1:91,1] = PR[GP1:90,1] + 67.822;
   1:  PR[GP1:91,2] = PR[GP1:90,2] + 11.294;
   1:L PR[91] 10mm/sec CNT100;
   1:  PR[GP1:91,1] = PR[GP1:90,1] + 65.168;
   1:  PR[GP1:91,2] = PR[GP1:90,2] + 16.581;
   1:L PR[91] 10mm/sec CNT100;
   1:  PR[GP1:91,1] = PR[GP1:90,1] + 63.797;
   1:  PR[GP1:91,2] = PR[GP1:90,2] + 19.262;
   1:L PR[91] 10mm/sec CNT100;
   1:  PR[GP1:91,1] = PR[GP1:90,1] + 61.681;
   1:  PR[GP1:91,2] = PR[GP1:90,2] + 22.001;
   1:L PR[91] 10mm/sec CNT100;
   1:  PR[GP1:91,1] = PR[GP1:90,1] + 58.451;
   1:  PR[GP1:91,2] = PR[GP1:90,2] + 25.407;
   1:L PR[91] 10mm/sec CNT100;
   1:  PR[GP1:91,1] = PR[GP1:90,1] + 55.502;
   1:  PR[GP1:91,2] = PR[GP1:90,2] + 28.042;
   1:L PR[91] 10mm/sec CNT100;
   1:  PR[GP1:91,1] = PR[GP1:90,1] + 52.786;
   1:  PR[GP1:91,2] = PR[GP1:90,2] + 29.569;
   1:L PR[91] 10mm/sec CNT100;
   1:  PR[GP1:91,1] = PR[GP1:90,1] + 48.960;
   1:  PR[GP1:91,2] = PR[GP1:90,2] + 31.980;
   1:L PR[91] 10mm/sec CNT100;
   1:  PR[GP1:91,1] = PR[GP1:90,1] + 43.352;
   1:  PR[GP1:91,2] = PR[GP1:90,2] + 34.175;
   1:L PR[91] 10mm/sec CNT100;
   1:  PR[GP1:91,1] = PR[GP1:90,1] + 36.576;
   1:  PR[GP1:91,2] = PR[GP1:90,2] + 35.635;
   1:L PR[91] 10mm/sec CNT100;
   1:  PR[GP1:91,1] = PR[GP1:90,1] + 30.484;
   1:  PR[GP1:91,2] = PR[GP1:90,2] + 35.865;
   1:L PR[91] 10mm/sec CNT100;
   1:  PR[GP1:91,1] = PR[GP1:90,1] + 28.987;
   1:  PR[GP1:91,2] = PR[GP1:90,2] + 35.870;
   1:L PR[91] 10mm/sec CNT100;
   1:  PR[GP1:91,1] = PR[GP1:90,1] + 23.032;
   1:  PR[GP1:91,2] = PR[GP1:90,2] + 35.087;
   1:L PR[91] 10mm/sec CNT100;
   1:  PR[GP1:91,1] = PR[GP1:90,1] + 17.928;
   1:  PR[GP1:91,2] = PR[GP1:90,2] + 33.463;
   1:L PR[91] 10mm/sec CNT100;
   1:  PR[GP1:91,1] = PR[GP1:90,1] + 15.089;
   1:  PR[GP1:91,2] = PR[GP1:90,2] + 32.479;
   1:L PR[91] 10mm/sec CNT100;
   1:  PR[GP1:91,1] = PR[GP1:90,1] + 10.523;
   1:  PR[GP1:91,2] = PR[GP1:90,2] + 30.096;
   1:L PR[91] 10mm/sec CNT100;
   1:  PR[GP1:91,1] = PR[GP1:90,1] + 9.019;
   1:  PR[GP1:91,2] = PR[GP1:90,2] + 29.033;
   1:L PR[91] 10mm/sec CNT100;
   1:  PR[GP1:91,1] = PR[GP1:90,1] + 6.229;
   1:  PR[GP1:91,2] = PR[GP1:90,2] + 26.851;
   1:L PR[91] 10mm/sec CNT100;
   1:  PR[GP1:91,1] = PR[GP1:90,1] + 4.066;
   1:  PR[GP1:91,2] = PR[GP1:90,2] + 24.334;
   1:L PR[91] 10mm/sec CNT100;
   1:  PR[GP1:91,1] = PR[GP1:90,1] + 2.958;
   1:  PR[GP1:91,2] = PR[GP1:90,2] + 23.896;
   1:L PR[91] 10mm/sec CNT100;
   1:  PR[GP1:91,1] = PR[GP1:90,1] + 1.156;
   1:  PR[GP1:91,2] = PR[GP1:90,2] + 22.975;
   1:L PR[91] 10mm/sec CNT100;
   1:  PR[GP1:91,1] = PR[GP1:90,1] + -1.314;
   1:  PR[GP1:91,2] = PR[GP1:90,2] + 24.023;
   1:  PR[GP1:91,3] = PR[GP1:90,3] + 49.210;
   1:L PR[91] 10mm/sec CNT100;
   1:  PR[GP1:91,1] = PR[GP1:90,1] + -3.197;
   1:  PR[GP1:91,2] = PR[GP1:90,2] + 24.981;
   1:L PR[91] 10mm/sec CNT100;
   1:  PR[GP1:91,1] = PR[GP1:90,1] + -5.045;
   1:  PR[GP1:91,2] = PR[GP1:90,2] + 27.130;
   1:L PR[91] 10mm/sec CNT100;
   1:  PR[GP1:91,1] = PR[GP1:90,1] + -7.469;
   1:  PR[GP1:91,2] = PR[GP1:90,2] + 29.028;
   1:L PR[91] 10mm/sec CNT100;
   1:  PR[GP1:91,1] = PR[GP1:90,1] + -9.230;
   1:  PR[GP1:91,2] = PR[GP1:90,2] + 30.272;
   1:L PR[91] 10mm/sec CNT100;
   1:  PR[GP1:91,1] = PR[GP1:90,1] + -13.532;
   1:  PR[GP1:91,2] = PR[GP1:90,2] + 32.523;
   1:L PR[91] 10mm/sec CNT100;
   1:  PR[GP1:91,1] = PR[GP1:90,1] + -18.807;
   1:  PR[GP1:91,2] = PR[GP1:90,2] + 34.218;
   1:L PR[91] 10mm/sec CNT100;
   1:  PR[GP1:91,1] = PR[GP1:90,1] + -21.791;
   1:  PR[GP1:91,2] = PR[GP1:90,2] + 35.249;
   1:L PR[91] 10mm/sec CNT100;
   1:  PR[GP1:91,1] = PR[GP1:90,1] + -27.404;
   1:  PR[GP1:91,2] = PR[GP1:90,2] + 35.983;
   1:L PR[91] 10mm/sec CNT100;
   1:  PR[GP1:91,1] = PR[GP1:90,1] + -33.959;
   1:  PR[GP1:91,2] = PR[GP1:90,2] + 35.757;
   1:L PR[91] 10mm/sec CNT100;
   1:  PR[GP1:91,1] = PR[GP1:90,1] + -35.398;
   1:  PR[GP1:91,2] = PR[GP1:90,2] + 35.750;
   1:L PR[91] 10mm/sec CNT100;
   1:  PR[GP1:91,1] = PR[GP1:90,1] + -41.799;
   1:  PR[GP1:91,2] = PR[GP1:90,2] + 34.369;
   1:L PR[91] 10mm/sec CNT100;
   1:  PR[GP1:91,1] = PR[GP1:90,1] + -48.187;
   1:  PR[GP1:91,2] = PR[GP1:90,2] + 31.846;
   1:L PR[91] 10mm/sec CNT100;
   1:  PR[GP1:91,1] = PR[GP1:90,1] + -48.803;
   1:  PR[GP1:91,2] = PR[GP1:90,2] + 31.495;
   1:L PR[91] 10mm/sec CNT100;
   1:  PR[GP1:91,1] = PR[GP1:90,1] + -54.251;
   1:  PR[GP1:91,2] = PR[GP1:90,2] + 28.120;
   1:L PR[91] 10mm/sec CNT100;
   1:  PR[GP1:91,1] = PR[GP1:90,1] + -57.798;
   1:  PR[GP1:91,2] = PR[GP1:90,2] + 24.941;
   1:L PR[91] 10mm/sec CNT100;
   1:  PR[GP1:91,1] = PR[GP1:90,1] + -60.109;
   1:  PR[GP1:91,2] = PR[GP1:90,2] + 22.511;
   1:L PR[91] 10mm/sec CNT100;
   1:  PR[GP1:91,1] = PR[GP1:90,1] + -62.722;
   1:  PR[GP1:91,2] = PR[GP1:90,2] + 19.120;
   1:L PR[91] 10mm/sec CNT100;
   1:  PR[GP1:91,1] = PR[GP1:90,1] + -66.540;
   1:  PR[GP1:91,2] = PR[GP1:90,2] + 11.516;
   1:L PR[91] 10mm/sec CNT100;
   1:  PR[GP1:91,1] = PR[GP1:90,1] + -67.465;
   1:  PR[GP1:91,2] = PR[GP1:90,2] + 8.375;
   1:L PR[91] 10mm/sec CNT100;
   1:  PR[GP1:91,1] = PR[GP1:90,1] + -68.296;
   1:  PR[GP1:91,2] = PR[GP1:90,2] + 3.046;
   1:L PR[91] 10mm/sec CNT100;
   1:  PR[GP1:91,1] = PR[GP1:90,1] + -68.568;
   1:  PR[GP1:91,2] = PR[GP1:90,2] + 0.016;
   1:L PR[91] 10mm/sec CNT100;
   1:  PR[GP1:91,1] = PR[GP1:90,1] + -67.740;
   1:  PR[GP1:91,2] = PR[GP1:90,2] + -5.225;
   1:L PR[91] 10mm/sec CNT100;
   1:  PR[GP1:91,1] = PR[GP1:90,1] + -67.459;
   1:  PR[GP1:91,2] = PR[GP1:90,2] + -8.404;
   1:L PR[91] 10mm/sec CNT100;
   1:  PR[GP1:91,1] = PR[GP1:90,1] + -66.540;
   1:  PR[GP1:91,2] = PR[GP1:90,2] + -11.525;
   1:L PR[91] 10mm/sec CNT100;
   1:  PR[GP1:91,1] = PR[GP1:90,1] + -62.722;
   1:  PR[GP1:91,2] = PR[GP1:90,2] + -19.129;
   1:L PR[91] 10mm/sec CNT100;
   1:  PR[GP1:91,1] = PR[GP1:90,1] + -60.109;
   1:  PR[GP1:91,2] = PR[GP1:90,2] + -22.520;
   1:L PR[91] 10mm/sec CNT100;
   1:  PR[GP1:91,1] = PR[GP1:90,1] + -57.798;
   1:  PR[GP1:91,2] = PR[GP1:90,2] + -24.950;
   1:L PR[91] 10mm/sec CNT100;
   1:  PR[GP1:91,1] = PR[GP1:90,1] + -54.261;
   1:  PR[GP1:91,2] = PR[GP1:90,2] + -28.121;
   1:L PR[91] 10mm/sec CNT100;
   1:  PR[GP1:91,1] = PR[GP1:90,1] + -52.604;
   1:  PR[GP1:91,2] = PR[GP1:90,2] + -29.053;
   1:L PR[91] 10mm/sec CNT100;
   1:  PR[GP1:91,1] = PR[GP1:90,1] + -48.174;
   1:  PR[GP1:91,2] = PR[GP1:90,2] + -31.859;
   1:L PR[91] 10mm/sec CNT100;
   1:  PR[GP1:91,1] = PR[GP1:90,1] + -45.873;
   1:  PR[GP1:91,2] = PR[GP1:90,2] + -32.765;
   1:L PR[91] 10mm/sec CNT100;
   1:  PR[GP1:91,1] = PR[GP1:90,1] + -42.240;
   1:  PR[GP1:91,2] = PR[GP1:90,2] + -34.224;
   1:L PR[91] 10mm/sec CNT100;
   1:  PR[GP1:91,1] = PR[GP1:90,1] + -41.809;
   1:  PR[GP1:91,2] = PR[GP1:90,2] + -34.376;
   1:L PR[91] 10mm/sec CNT100;
   1:  PR[GP1:91,1] = PR[GP1:90,1] + -35.386;
   1:  PR[GP1:91,2] = PR[GP1:90,2] + -35.762;
   1:L PR[91] 10mm/sec CNT100;
   1:  PR[GP1:91,1] = PR[GP1:90,1] + -29.574;
   1:  PR[GP1:91,2] = PR[GP1:90,2] + -35.985;
   1:L PR[91] 10mm/sec CNT100;
   1:  PR[GP1:91,1] = PR[GP1:90,1] + -27.410;
   1:  PR[GP1:91,2] = PR[GP1:90,2] + -35.992;
   1:L PR[91] 10mm/sec CNT100;
   1:  PR[GP1:91,1] = PR[GP1:90,1] + -21.779;
   1:  PR[GP1:91,2] = PR[GP1:90,2] + -35.256;
   1:L PR[91] 10mm/sec CNT100;
   1:  PR[GP1:91,1] = PR[GP1:90,1] + -16.965;
   1:  PR[GP1:91,2] = PR[GP1:90,2] + -33.725;
   1:L PR[91] 10mm/sec CNT100;
   1:  PR[GP1:91,1] = PR[GP1:90,1] + -13.532;
   1:  PR[GP1:91,2] = PR[GP1:90,2] + -32.532;
   1:L PR[91] 10mm/sec CNT100;
   1:  PR[GP1:91,1] = PR[GP1:90,1] + -9.230;
   1:  PR[GP1:91,2] = PR[GP1:90,2] + -30.280;
   1:L PR[91] 10mm/sec CNT100;
   1:  PR[GP1:91,1] = PR[GP1:90,1] + -6.794;
   1:  PR[GP1:91,2] = PR[GP1:90,2] + -28.511;
   1:L PR[91] 10mm/sec CNT100;
   1:  PR[GP1:91,1] = PR[GP1:90,1] + -4.743;
   1:  PR[GP1:91,2] = PR[GP1:90,2] + -26.905;
   1:L PR[91] 10mm/sec CNT100;
   1:  PR[GP1:91,1] = PR[GP1:90,1] + -3.141;
   1:  PR[GP1:91,2] = PR[GP1:90,2] + -25.047;
   1:L PR[91] 10mm/sec CNT100;
   1:  PR[GP1:91,1] = PR[GP1:90,1] + -0.399;
   1:  PR[GP1:91,2] = PR[GP1:90,2] + -24.458;
   1:L PR[91] 10mm/sec CNT100;
   1:  PR[GP1:91,1] = PR[GP1:90,1] + 1.133;
   1:  PR[GP1:91,2] = PR[GP1:90,2] + -23.647;
   1:L PR[91] 10mm/sec CNT100;
   1:  PR[GP1:91,1] = PR[GP1:90,1] + 4.018;
   1:  PR[GP1:91,2] = PR[GP1:90,2] + -25.110;
   1:L PR[91] 10mm/sec CNT100;
   1:  PR[GP1:91,1] = PR[GP1:90,1] + 5.580;
   1:  PR[GP1:91,2] = PR[GP1:90,2] + -26.924;
   1:L PR[91] 10mm/sec CNT100;
   1:  PR[GP1:91,1] = PR[GP1:90,1] + 7.622;
   1:  PR[GP1:91,2] = PR[GP1:90,2] + -28.521;
   1:L PR[91] 10mm/sec CNT100;
   1:  PR[GP1:91,1] = PR[GP1:90,1] + 10.062;
   1:  PR[GP1:91,2] = PR[GP1:90,2] + -30.294;
   1:L PR[91] 10mm/sec CNT100;
   1:  PR[GP1:91,1] = PR[GP1:90,1] + 14.333;
   1:  PR[GP1:91,2] = PR[GP1:90,2] + -32.523;
   1:L PR[91] 10mm/sec CNT100;
   1:  PR[GP1:91,1] = PR[GP1:90,1] + 19.614;
   1:  PR[GP1:91,2] = PR[GP1:90,2] + -34.219;
   1:L PR[91] 10mm/sec CNT100;
   1:  PR[GP1:91,1] = PR[GP1:90,1] + 22.602;
   1:  PR[GP1:91,2] = PR[GP1:90,2] + -35.254;
   1:L PR[91] 10mm/sec CNT100;
   1:  PR[GP1:91,1] = PR[GP1:90,1] + 28.208;
   1:  PR[GP1:91,2] = PR[GP1:90,2] + -35.991;
   1:L PR[91] 10mm/sec CNT100;
   1:  PR[GP1:91,1] = PR[GP1:90,1] + 34.733;
   1:  PR[GP1:91,2] = PR[GP1:90,2] + -35.772;
   1:L PR[91] 10mm/sec CNT100;
   1:  PR[GP1:91,1] = PR[GP1:90,1] + 36.177;
   1:  PR[GP1:91,2] = PR[GP1:90,2] + -35.765;
   1:L PR[91] 10mm/sec CNT100;
   1:  PR[GP1:91,1] = PR[GP1:90,1] + 42.569;
   1:  PR[GP1:91,2] = PR[GP1:90,2] + -34.390;
   1:L PR[91] 10mm/sec CNT100;
   1:  PR[GP1:91,1] = PR[GP1:90,1] + 48.978;
   1:  PR[GP1:91,2] = PR[GP1:90,2] + -31.871;
   1:L PR[91] 10mm/sec CNT100;
   1:  PR[GP1:91,1] = PR[GP1:90,1] + 49.585;
   1:  PR[GP1:91,2] = PR[GP1:90,2] + -31.526;
   1:L PR[91] 10mm/sec CNT100;
   1:  PR[GP1:91,1] = PR[GP1:90,1] + 55.020;
   1:  PR[GP1:91,2] = PR[GP1:90,2] + -28.175;
   1:L PR[91] 10mm/sec CNT100;
   1:  PR[GP1:91,1] = PR[GP1:90,1] + 58.564;
   1:  PR[GP1:91,2] = PR[GP1:90,2] + -25.007;
   1:L PR[91] 10mm/sec CNT100;
   1:  PR[GP1:91,1] = PR[GP1:90,1] + 60.869;
   1:  PR[GP1:91,2] = PR[GP1:90,2] + -22.577;
   1:L PR[91] 10mm/sec CNT100;
   1:  PR[GP1:91,1] = PR[GP1:90,1] + 63.520;
   1:  PR[GP1:91,2] = PR[GP1:90,2] + -19.146;
   1:L PR[91] 10mm/sec CNT100;
   1:  PR[GP1:91,1] = PR[GP1:90,1] + 65.548;
   1:  PR[GP1:91,2] = PR[GP1:90,2] + -15.110;
   1:L PR[91] 10mm/sec CNT100;
   1:  PR[GP1:91,1] = PR[GP1:90,1] + 67.347;
   1:  PR[GP1:91,2] = PR[GP1:90,2] + -11.584;
   1:L PR[91] 10mm/sec CNT100;
   1:  PR[GP1:91,1] = PR[GP1:90,1] + 68.271;
   1:  PR[GP1:91,2] = PR[GP1:90,2] + -8.487;
   1:L PR[91] 10mm/sec CNT100;
   1:  PR[GP1:91,1] = PR[GP1:90,1] + 69.102;
   1:  PR[GP1:91,2] = PR[GP1:90,2] + -3.142;
   1:L PR[91] 10mm/sec CNT100;
   1:  PR[GP1:91,1] = PR[GP1:90,1] + 69.388;
   1:  PR[GP1:91,2] = PR[GP1:90,2] + -0.024;
   1:L PR[91] 10mm/sec CNT100;
   1:  PR[GP1:91,1] = PR[GP1:90,1] + 68.561;
   1:  PR[GP1:91,2] = PR[GP1:90,2] + 5.231;
   1:L PR[91] 10mm/sec CNT100;
   1:  PR[GP1:91,1] = PR[GP1:90,1] + 68.265;
   1:  PR[GP1:91,2] = PR[GP1:90,2] + 8.497;
   1:L PR[91] 10mm/sec CNT100;
   1:  PR[GP1:91,1] = PR[GP1:90,1] + 67.346;
   1:  PR[GP1:91,2] = PR[GP1:90,2] + 11.577;
   1:L PR[91] 10mm/sec CNT100;
   1:  PR[GP1:91,1] = PR[GP1:90,1] + 65.236;
   1:  PR[GP1:91,2] = PR[GP1:90,2] + 15.780;
   1:L PR[91] 10mm/sec CNT100;
   1:  PR[GP1:91,1] = PR[GP1:90,1] + 63.521;
   1:  PR[GP1:91,2] = PR[GP1:90,2] + 19.135;
   1:L PR[91] 10mm/sec CNT100;
   1:  PR[GP1:91,1] = PR[GP1:90,1] + 60.869;
   1:  PR[GP1:91,2] = PR[GP1:90,2] + 22.568;
   1:L PR[91] 10mm/sec CNT100;
   1:  PR[GP1:91,1] = PR[GP1:90,1] + 58.564;
   1:  PR[GP1:91,2] = PR[GP1:90,2] + 24.998;
   1:L PR[91] 10mm/sec CNT100;
   1:  PR[GP1:91,1] = PR[GP1:90,1] + 55.029;
   1:  PR[GP1:91,2] = PR[GP1:90,2] + 28.158;
   1:L PR[91] 10mm/sec CNT100;
   1:  PR[GP1:91,1] = PR[GP1:90,1] + 53.382;
   1:  PR[GP1:91,2] = PR[GP1:90,2] + 29.083;
   1:L PR[91] 10mm/sec CNT100;
   1:  PR[GP1:91,1] = PR[GP1:90,1] + 48.965;
   1:  PR[GP1:91,2] = PR[GP1:90,2] + 31.867;
   1:L PR[91] 10mm/sec CNT100;
   1:  PR[GP1:91,1] = PR[GP1:90,1] + 46.694;
   1:  PR[GP1:91,2] = PR[GP1:90,2] + 32.756;
   1:L PR[91] 10mm/sec CNT100;
   1:  PR[GP1:91,1] = PR[GP1:90,1] + 43.017;
   1:  PR[GP1:91,2] = PR[GP1:90,2] + 34.224;
   1:L PR[91] 10mm/sec CNT100;
   1:  PR[GP1:91,1] = PR[GP1:90,1] + 42.581;
   1:  PR[GP1:91,2] = PR[GP1:90,2] + 34.378;
   1:L PR[91] 10mm/sec CNT100;
   1:  PR[GP1:91,1] = PR[GP1:90,1] + 36.169;
   1:  PR[GP1:91,2] = PR[GP1:90,2] + 35.758;
   1:L PR[91] 10mm/sec CNT100;
   1:  PR[GP1:91,1] = PR[GP1:90,1] + 30.386;
   1:  PR[GP1:91,2] = PR[GP1:90,2] + 35.976;
   1:L PR[91] 10mm/sec CNT100;
   1:  PR[GP1:91,1] = PR[GP1:90,1] + 28.221;
   1:  PR[GP1:91,2] = PR[GP1:90,2] + 35.984;
   1:L PR[91] 10mm/sec CNT100;
   1:  PR[GP1:91,1] = PR[GP1:90,1] + 22.599;
   1:  PR[GP1:91,2] = PR[GP1:90,2] + 35.245;
   1:L PR[91] 10mm/sec CNT100;
   1:  PR[GP1:91,1] = PR[GP1:90,1] + 17.780;
   1:  PR[GP1:91,2] = PR[GP1:90,2] + 33.711;
   1:L PR[91] 10mm/sec CNT100;
   1:  PR[GP1:91,1] = PR[GP1:90,1] + 14.344;
   1:  PR[GP1:91,2] = PR[GP1:90,2] + 32.520;
   1:L PR[91] 10mm/sec CNT100;
   1:  PR[GP1:91,1] = PR[GP1:90,1] + 10.063;
   1:  PR[GP1:91,2] = PR[GP1:90,2] + 30.286;
   1:L PR[91] 10mm/sec CNT100;
   1:  PR[GP1:91,1] = PR[GP1:90,1] + 8.298;
   1:  PR[GP1:91,2] = PR[GP1:90,2] + 29.039;
   1:L PR[91] 10mm/sec CNT100;
   1:  PR[GP1:91,1] = PR[GP1:90,1] + 5.885;
   1:  PR[GP1:91,2] = PR[GP1:90,2] + 27.152;
   1:L PR[91] 10mm/sec CNT100;
   1:  PR[GP1:91,1] = PR[GP1:90,1] + 4.001;
   1:  PR[GP1:91,2] = PR[GP1:90,2] + 24.959;
   1:L PR[91] 10mm/sec CNT100;
   1:  PR[GP1:91,1] = PR[GP1:90,1] + 2.765;
   1:  PR[GP1:91,2] = PR[GP1:90,2] + 24.470;
   1:L PR[91] 10mm/sec CNT100;
   1:  PR[GP1:91,1] = PR[GP1:90,1] + 1.246;
   1:  PR[GP1:91,2] = PR[GP1:90,2] + 23.694;
   1:L PR[91] 10mm/sec CNT100;
   1:  PR[GP1:91,1] = PR[GP1:90,1] + -1.508;
   1:  PR[GP1:91,2] = PR[GP1:90,2] + 24.779;
   1:  PR[GP1:91,3] = PR[GP1:90,3] + 50.540;
   1:L PR[91] 10mm/sec CNT100;
   1:  PR[GP1:91,1] = PR[GP1:90,1] + -3.134;
   1:  PR[GP1:91,2] = PR[GP1:90,2] + 25.606;
   1:L PR[91] 10mm/sec CNT100;
   1:  PR[GP1:91,1] = PR[GP1:90,1] + -4.705;
   1:  PR[GP1:91,2] = PR[GP1:90,2] + 27.434;
   1:L PR[91] 10mm/sec CNT100;
   1:  PR[GP1:91,1] = PR[GP1:90,1] + -6.750;
   1:  PR[GP1:91,2] = PR[GP1:90,2] + 29.035;
   1:L PR[91] 10mm/sec CNT100;
   1:  PR[GP1:91,1] = PR[GP1:90,1] + -8.770;
   1:  PR[GP1:91,2] = PR[GP1:90,2] + 30.462;
   1:L PR[91] 10mm/sec CNT100;
   1:  PR[GP1:91,1] = PR[GP1:90,1] + -12.787;
   1:  PR[GP1:91,2] = PR[GP1:90,2] + 32.564;
   1:L PR[91] 10mm/sec CNT100;
   1:  PR[GP1:91,1] = PR[GP1:90,1] + -17.715;
   1:  PR[GP1:91,2] = PR[GP1:90,2] + 34.147;
   1:L PR[91] 10mm/sec CNT100;
   1:  PR[GP1:91,1] = PR[GP1:90,1] + -21.359;
   1:  PR[GP1:91,2] = PR[GP1:90,2] + 35.407;
   1:L PR[91] 10mm/sec CNT100;
   1:  PR[GP1:91,1] = PR[GP1:90,1] + -26.638;
   1:  PR[GP1:91,2] = PR[GP1:90,2] + 36.097;
   1:L PR[91] 10mm/sec CNT100;
   1:  PR[GP1:91,1] = PR[GP1:90,1] + -32.808;
   1:  PR[GP1:91,2] = PR[GP1:90,2] + 35.885;
   1:L PR[91] 10mm/sec CNT100;
   1:  PR[GP1:91,1] = PR[GP1:90,1] + -34.988;
   1:  PR[GP1:91,2] = PR[GP1:90,2] + 35.874;
   1:L PR[91] 10mm/sec CNT100;
   1:  PR[GP1:91,1] = PR[GP1:90,1] + -41.045;
   1:  PR[GP1:91,2] = PR[GP1:90,2] + 34.567;
   1:L PR[91] 10mm/sec CNT100;
   1:  PR[GP1:91,1] = PR[GP1:90,1] + -47.660;
   1:  PR[GP1:91,2] = PR[GP1:90,2] + 31.948;
   1:L PR[91] 10mm/sec CNT100;
   1:  PR[GP1:91,1] = PR[GP1:90,1] + -47.983;
   1:  PR[GP1:91,2] = PR[GP1:90,2] + 31.833;
   1:L PR[91] 10mm/sec CNT100;
   1:  PR[GP1:91,1] = PR[GP1:90,1] + -53.786;
   1:  PR[GP1:91,2] = PR[GP1:90,2] + 28.229;
   1:L PR[91] 10mm/sec CNT100;
   1:  PR[GP1:91,1] = PR[GP1:90,1] + -57.920;
   1:  PR[GP1:91,2] = PR[GP1:90,2] + 24.524;
   1:L PR[91] 10mm/sec CNT100;
   1:  PR[GP1:91,1] = PR[GP1:90,1] + -59.309;
   1:  PR[GP1:91,2] = PR[GP1:90,2] + 23.063;
   1:L PR[91] 10mm/sec CNT100;
   1:  PR[GP1:91,1] = PR[GP1:90,1] + -62.450;
   1:  PR[GP1:91,2] = PR[GP1:90,2] + 18.986;
   1:L PR[91] 10mm/sec CNT100;
   1:  PR[GP1:91,1] = PR[GP1:90,1] + -66.067;
   1:  PR[GP1:91,2] = PR[GP1:90,2] + 11.791;
   1:L PR[91] 10mm/sec CNT100;
   1:  PR[GP1:91,1] = PR[GP1:90,1] + -67.210;
   1:  PR[GP1:91,2] = PR[GP1:90,2] + 7.909;
   1:L PR[91] 10mm/sec CNT100;
   1:  PR[GP1:91,1] = PR[GP1:90,1] + -67.845;
   1:  PR[GP1:91,2] = PR[GP1:90,2] + 3.838;
   1:L PR[91] 10mm/sec CNT100;
   1:  PR[GP1:91,1] = PR[GP1:90,1] + -68.189;
   1:  PR[GP1:91,2] = PR[GP1:90,2] + 0.016;
   1:L PR[91] 10mm/sec CNT100;
   1:  PR[GP1:91,1] = PR[GP1:90,1] + -67.551;
   1:  PR[GP1:91,2] = PR[GP1:90,2] + -4.019;
   1:L PR[91] 10mm/sec CNT100;
   1:  PR[GP1:91,1] = PR[GP1:90,1] + -67.205;
   1:  PR[GP1:91,2] = PR[GP1:90,2] + -7.937;
   1:L PR[91] 10mm/sec CNT100;
   1:  PR[GP1:91,1] = PR[GP1:90,1] + -66.067;
   1:  PR[GP1:91,2] = PR[GP1:90,2] + -11.800;
   1:L PR[91] 10mm/sec CNT100;
   1:  PR[GP1:91,1] = PR[GP1:90,1] + -62.450;
   1:  PR[GP1:91,2] = PR[GP1:90,2] + -18.995;
   1:L PR[91] 10mm/sec CNT100;
   1:  PR[GP1:91,1] = PR[GP1:90,1] + -59.309;
   1:  PR[GP1:91,2] = PR[GP1:90,2] + -23.072;
   1:L PR[91] 10mm/sec CNT100;
   1:  PR[GP1:91,1] = PR[GP1:90,1] + -57.920;
   1:  PR[GP1:91,2] = PR[GP1:90,2] + -24.533;
   1:L PR[91] 10mm/sec CNT100;
   1:  PR[GP1:91,1] = PR[GP1:90,1] + -53.796;
   1:  PR[GP1:91,2] = PR[GP1:90,2] + -28.229;
   1:L PR[91] 10mm/sec CNT100;
   1:  PR[GP1:91,1] = PR[GP1:90,1] + -53.206;
   1:  PR[GP1:91,2] = PR[GP1:90,2] + -28.561;
   1:L PR[91] 10mm/sec CNT100;
   1:  PR[GP1:91,1] = PR[GP1:90,1] + -50.653;
   1:  PR[GP1:91,2] = PR[GP1:90,2] + -30.179;
   1:L PR[91] 10mm/sec CNT100;
   1:  PR[GP1:91,1] = PR[GP1:90,1] + -47.972;
   1:  PR[GP1:91,2] = PR[GP1:90,2] + -31.849;
   1:L PR[91] 10mm/sec CNT100;
   1:  PR[GP1:91,1] = PR[GP1:90,1] + -42.140;
   1:  PR[GP1:91,2] = PR[GP1:90,2] + -34.191;
   1:L PR[91] 10mm/sec CNT100;
   1:  PR[GP1:91,1] = PR[GP1:90,1] + -41.055;
   1:  PR[GP1:91,2] = PR[GP1:90,2] + -34.574;
   1:L PR[91] 10mm/sec CNT100;
   1:  PR[GP1:91,1] = PR[GP1:90,1] + -34.976;
   1:  PR[GP1:91,2] = PR[GP1:90,2] + -35.885;
   1:L PR[91] 10mm/sec CNT100;
   1:  PR[GP1:91,1] = PR[GP1:90,1] + -29.474;
   1:  PR[GP1:91,2] = PR[GP1:90,2] + -36.097;
   1:L PR[91] 10mm/sec CNT100;
   1:  PR[GP1:91,1] = PR[GP1:90,1] + -26.642;
   1:  PR[GP1:91,2] = PR[GP1:90,2] + -36.106;
   1:L PR[91] 10mm/sec CNT100;
   1:  PR[GP1:91,1] = PR[GP1:90,1] + -21.345;
   1:  PR[GP1:91,2] = PR[GP1:90,2] + -35.414;
   1:L PR[91] 10mm/sec CNT100;
   1:  PR[GP1:91,1] = PR[GP1:90,1] + -16.816;
   1:  PR[GP1:91,2] = PR[GP1:90,2] + -33.973;
   1:L PR[91] 10mm/sec CNT100;
   1:  PR[GP1:91,1] = PR[GP1:90,1] + -12.786;
   1:  PR[GP1:91,2] = PR[GP1:90,2] + -32.572;
   1:L PR[91] 10mm/sec CNT100;
   1:  PR[GP1:91,1] = PR[GP1:90,1] + -8.770;
   1:  PR[GP1:91,2] = PR[GP1:90,2] + -30.470;
   1:L PR[91] 10mm/sec CNT100;
   1:  PR[GP1:91,1] = PR[GP1:90,1] + -5.978;
   1:  PR[GP1:91,2] = PR[GP1:90,2] + -28.442;
   1:L PR[91] 10mm/sec CNT100;
   1:  PR[GP1:91,1] = PR[GP1:90,1] + -4.365;
   1:  PR[GP1:91,2] = PR[GP1:90,2] + -27.179;
   1:L PR[91] 10mm/sec CNT100;
   1:  PR[GP1:91,1] = PR[GP1:90,1] + -3.077;
   1:  PR[GP1:91,2] = PR[GP1:90,2] + -25.685;
   1:L PR[91] 10mm/sec CNT100;
   1:  PR[GP1:91,1] = PR[GP1:90,1] + -0.035;
   1:  PR[GP1:91,2] = PR[GP1:90,2] + -25.032;
   1:L PR[91] 10mm/sec CNT100;
   1:  PR[GP1:91,1] = PR[GP1:90,1] + 1.222;
   1:  PR[GP1:91,2] = PR[GP1:90,2] + -24.366;
   1:L PR[91] 10mm/sec CNT100;
   1:  PR[GP1:91,1] = PR[GP1:90,1] + 3.953;
   1:  PR[GP1:91,2] = PR[GP1:90,2] + -25.749;
   1:L PR[91] 10mm/sec CNT100;
   1:  PR[GP1:91,1] = PR[GP1:90,1] + 5.198;
   1:  PR[GP1:91,2] = PR[GP1:90,2] + -27.195;
   1:L PR[91] 10mm/sec CNT100;
   1:  PR[GP1:91,1] = PR[GP1:90,1] + 6.803;
   1:  PR[GP1:91,2] = PR[GP1:90,2] + -28.451;
   1:L PR[91] 10mm/sec CNT100;
   1:  PR[GP1:91,1] = PR[GP1:90,1] + 9.601;
   1:  PR[GP1:91,2] = PR[GP1:90,2] + -30.483;
   1:L PR[91] 10mm/sec CNT100;
   1:  PR[GP1:91,1] = PR[GP1:90,1] + 13.587;
   1:  PR[GP1:91,2] = PR[GP1:90,2] + -32.563;
   1:L PR[91] 10mm/sec CNT100;
   1:  PR[GP1:91,1] = PR[GP1:90,1] + 18.520;
   1:  PR[GP1:91,2] = PR[GP1:90,2] + -34.148;
   1:L PR[91] 10mm/sec CNT100;
   1:  PR[GP1:91,1] = PR[GP1:90,1] + 22.169;
   1:  PR[GP1:91,2] = PR[GP1:90,2] + -35.412;
   1:L PR[91] 10mm/sec CNT100;
   1:  PR[GP1:91,1] = PR[GP1:90,1] + 27.441;
   1:  PR[GP1:91,2] = PR[GP1:90,2] + -36.105;
   1:L PR[91] 10mm/sec CNT100;
   1:  PR[GP1:91,1] = PR[GP1:90,1] + 33.582;
   1:  PR[GP1:91,2] = PR[GP1:90,2] + -35.898;
   1:L PR[91] 10mm/sec CNT100;
   1:  PR[GP1:91,1] = PR[GP1:90,1] + 35.769;
   1:  PR[GP1:91,2] = PR[GP1:90,2] + -35.889;
   1:L PR[91] 10mm/sec CNT100;
   1:  PR[GP1:91,1] = PR[GP1:90,1] + 41.817;
   1:  PR[GP1:91,2] = PR[GP1:90,2] + -34.587;
   1:L PR[91] 10mm/sec CNT100;
   1:  PR[GP1:91,1] = PR[GP1:90,1] + 48.441;
   1:  PR[GP1:91,2] = PR[GP1:90,2] + -31.977;
   1:L PR[91] 10mm/sec CNT100;
   1:  PR[GP1:91,1] = PR[GP1:90,1] + 48.770;
   1:  PR[GP1:91,2] = PR[GP1:90,2] + -31.861;
   1:L PR[91] 10mm/sec CNT100;
   1:  PR[GP1:91,1] = PR[GP1:90,1] + 54.546;
   1:  PR[GP1:91,2] = PR[GP1:90,2] + -28.290;
   1:L PR[91] 10mm/sec CNT100;
   1:  PR[GP1:91,1] = PR[GP1:90,1] + 58.677;
   1:  PR[GP1:91,2] = PR[GP1:90,2] + -24.599;
   1:L PR[91] 10mm/sec CNT100;
   1:  PR[GP1:91,1] = PR[GP1:90,1] + 60.056;
   1:  PR[GP1:91,2] = PR[GP1:90,2] + -23.144;
   1:L PR[91] 10mm/sec CNT100;
   1:  PR[GP1:91,1] = PR[GP1:90,1] + 63.243;
   1:  PR[GP1:91,2] = PR[GP1:90,2] + -19.019;
   1:L PR[91] 10mm/sec CNT100;
   1:  PR[GP1:91,1] = PR[GP1:90,1] + 64.653;
   1:  PR[GP1:91,2] = PR[GP1:90,2] + -16.214;
   1:L PR[91] 10mm/sec CNT100;
   1:  PR[GP1:91,1] = PR[GP1:90,1] + 66.871;
   1:  PR[GP1:91,2] = PR[GP1:90,2] + -11.867;
   1:L PR[91] 10mm/sec CNT100;
   1:  PR[GP1:91,1] = PR[GP1:90,1] + 68.014;
   1:  PR[GP1:91,2] = PR[GP1:90,2] + -8.037;
   1:L PR[91] 10mm/sec CNT100;
   1:  PR[GP1:91,1] = PR[GP1:90,1] + 68.648;
   1:  PR[GP1:91,2] = PR[GP1:90,2] + -3.957;
   1:L PR[91] 10mm/sec CNT100;
   1:  PR[GP1:91,1] = PR[GP1:90,1] + 69.009;
   1:  PR[GP1:91,2] = PR[GP1:90,2] + -0.024;
   1:L PR[91] 10mm/sec CNT100;
   1:  PR[GP1:91,1] = PR[GP1:90,1] + 68.372;
   1:  PR[GP1:91,2] = PR[GP1:90,2] + 4.021;
   1:L PR[91] 10mm/sec CNT100;
   1:  PR[GP1:91,1] = PR[GP1:90,1] + 68.008;
   1:  PR[GP1:91,2] = PR[GP1:90,2] + 8.047;
   1:L PR[91] 10mm/sec CNT100;
   1:  PR[GP1:91,1] = PR[GP1:90,1] + 66.870;
   1:  PR[GP1:91,2] = PR[GP1:90,2] + 11.861;
   1:L PR[91] 10mm/sec CNT100;
   1:  PR[GP1:91,1] = PR[GP1:90,1] + 65.305;
   1:  PR[GP1:91,2] = PR[GP1:90,2] + 14.978;
   1:L PR[91] 10mm/sec CNT100;
   1:  PR[GP1:91,1] = PR[GP1:90,1] + 63.244;
   1:  PR[GP1:91,2] = PR[GP1:90,2] + 19.009;
   1:L PR[91] 10mm/sec CNT100;
   1:  PR[GP1:91,1] = PR[GP1:90,1] + 60.056;
   1:  PR[GP1:91,2] = PR[GP1:90,2] + 23.135;
   1:L PR[91] 10mm/sec CNT100;
   1:  PR[GP1:91,1] = PR[GP1:90,1] + 58.677;
   1:  PR[GP1:91,2] = PR[GP1:90,2] + 24.590;
   1:L PR[91] 10mm/sec CNT100;
   1:  PR[GP1:91,1] = PR[GP1:90,1] + 54.555;
   1:  PR[GP1:91,2] = PR[GP1:90,2] + 28.273;
   1:L PR[91] 10mm/sec CNT100;
   1:  PR[GP1:91,1] = PR[GP1:90,1] + 53.977;
   1:  PR[GP1:91,2] = PR[GP1:90,2] + 28.598;
   1:L PR[91] 10mm/sec CNT100;
   1:  PR[GP1:91,1] = PR[GP1:90,1] + 51.474;
   1:  PR[GP1:91,2] = PR[GP1:90,2] + 30.175;
   1:L PR[91] 10mm/sec CNT100;
   1:  PR[GP1:91,1] = PR[GP1:90,1] + 48.759;
   1:  PR[GP1:91,2] = PR[GP1:90,2] + 31.858;
   1:L PR[91] 10mm/sec CNT100;
   1:  PR[GP1:91,1] = PR[GP1:90,1] + 42.920;
   1:  PR[GP1:91,2] = PR[GP1:90,2] + 34.190;
   1:L PR[91] 10mm/sec CNT100;
   1:  PR[GP1:91,1] = PR[GP1:90,1] + 41.829;
   1:  PR[GP1:91,2] = PR[GP1:90,2] + 34.575;
   1:L PR[91] 10mm/sec CNT100;
   1:  PR[GP1:91,1] = PR[GP1:90,1] + 35.761;
   1:  PR[GP1:91,2] = PR[GP1:90,2] + 35.881;
   1:L PR[91] 10mm/sec CNT100;
   1:  PR[GP1:91,1] = PR[GP1:90,1] + 30.287;
   1:  PR[GP1:91,2] = PR[GP1:90,2] + 36.088;
   1:L PR[91] 10mm/sec CNT100;
   1:  PR[GP1:91,1] = PR[GP1:90,1] + 27.455;
   1:  PR[GP1:91,2] = PR[GP1:90,2] + 36.098;
   1:L PR[91] 10mm/sec CNT100;
   1:  PR[GP1:91,1] = PR[GP1:90,1] + 22.167;
   1:  PR[GP1:91,2] = PR[GP1:90,2] + 35.403;
   1:L PR[91] 10mm/sec CNT100;
   1:  PR[GP1:91,1] = PR[GP1:90,1] + 17.632;
   1:  PR[GP1:91,2] = PR[GP1:90,2] + 33.960;
   1:L PR[91] 10mm/sec CNT100;
   1:  PR[GP1:91,1] = PR[GP1:90,1] + 13.600;
   1:  PR[GP1:91,2] = PR[GP1:90,2] + 32.562;
   1:L PR[91] 10mm/sec CNT100;
   1:  PR[GP1:91,1] = PR[GP1:90,1] + 9.602;
   1:  PR[GP1:91,2] = PR[GP1:90,2] + 30.475;
   1:L PR[91] 10mm/sec CNT100;
   1:  PR[GP1:91,1] = PR[GP1:90,1] + 7.577;
   1:  PR[GP1:91,2] = PR[GP1:90,2] + 29.045;
   1:L PR[91] 10mm/sec CNT100;
   1:  PR[GP1:91,1] = PR[GP1:90,1] + 5.542;
   1:  PR[GP1:91,2] = PR[GP1:90,2] + 27.452;
   1:L PR[91] 10mm/sec CNT100;
   1:  PR[GP1:91,1] = PR[GP1:90,1] + 3.936;
   1:  PR[GP1:91,2] = PR[GP1:90,2] + 25.584;
   1:L PR[91] 10mm/sec CNT100;
   1:  PR[GP1:91,1] = PR[GP1:90,1] + 2.571;
   1:  PR[GP1:91,2] = PR[GP1:90,2] + 25.045;
   1:L PR[91] 10mm/sec CNT100;
   1:  PR[GP1:91,1] = PR[GP1:90,1] + 1.336;
   1:  PR[GP1:91,2] = PR[GP1:90,2] + 24.414;
   1:L PR[91] 10mm/sec CNT100;
   1:  PR[GP1:91,1] = PR[GP1:90,1] + -1.701;
   1:  PR[GP1:91,2] = PR[GP1:90,2] + 25.535;
   1:  PR[GP1:91,3] = PR[GP1:90,3] + 51.870;
   1:L PR[91] 10mm/sec CNT100;
   1:  PR[GP1:91,1] = PR[GP1:90,1] + -3.070;
   1:  PR[GP1:91,2] = PR[GP1:90,2] + 26.231;
   1:L PR[91] 10mm/sec CNT100;
   1:  PR[GP1:91,1] = PR[GP1:90,1] + -4.366;
   1:  PR[GP1:91,2] = PR[GP1:90,2] + 27.738;
   1:L PR[91] 10mm/sec CNT100;
   1:  PR[GP1:91,1] = PR[GP1:90,1] + -6.032;
   1:  PR[GP1:91,2] = PR[GP1:90,2] + 29.043;
   1:L PR[91] 10mm/sec CNT100;
   1:  PR[GP1:91,1] = PR[GP1:90,1] + -8.311;
   1:  PR[GP1:91,2] = PR[GP1:90,2] + 30.653;
   1:L PR[91] 10mm/sec CNT100;
   1:  PR[GP1:91,1] = PR[GP1:90,1] + -12.041;
   1:  PR[GP1:91,2] = PR[GP1:90,2] + 32.605;
   1:L PR[91] 10mm/sec CNT100;
   1:  PR[GP1:91,1] = PR[GP1:90,1] + -16.623;
   1:  PR[GP1:91,2] = PR[GP1:90,2] + 34.077;
   1:L PR[91] 10mm/sec CNT100;
   1:  PR[GP1:91,1] = PR[GP1:90,1] + -20.926;
   1:  PR[GP1:91,2] = PR[GP1:90,2] + 35.564;
   1:L PR[91] 10mm/sec CNT100;
   1:  PR[GP1:91,1] = PR[GP1:90,1] + -25.871;
   1:  PR[GP1:91,2] = PR[GP1:90,2] + 36.211;
   1:L PR[91] 10mm/sec CNT100;
   1:  PR[GP1:91,1] = PR[GP1:90,1] + -31.656;
   1:  PR[GP1:91,2] = PR[GP1:90,2] + 36.012;
   1:L PR[91] 10mm/sec CNT100;
   1:  PR[GP1:91,1] = PR[GP1:90,1] + -34.579;
   1:  PR[GP1:91,2] = PR[GP1:90,2] + 35.997;
   1:L PR[91] 10mm/sec CNT100;
   1:  PR[GP1:91,1] = PR[GP1:90,1] + -40.292;
   1:  PR[GP1:91,2] = PR[GP1:90,2] + 34.765;
   1:L PR[91] 10mm/sec CNT100;
   1:  PR[GP1:91,1] = PR[GP1:90,1] + -46.535;
   1:  PR[GP1:91,2] = PR[GP1:90,2] + 32.293;
   1:L PR[91] 10mm/sec CNT100;
   1:  PR[GP1:91,1] = PR[GP1:90,1] + -47.583;
   1:  PR[GP1:91,2] = PR[GP1:90,2] + 31.921;
   1:L PR[91] 10mm/sec CNT100;
   1:  PR[GP1:91,1] = PR[GP1:90,1] + -53.223;
   1:  PR[GP1:91,2] = PR[GP1:90,2] + 28.407;
   1:L PR[91] 10mm/sec CNT100;
   1:  PR[GP1:91,1] = PR[GP1:90,1] + -55.452;
   1:  PR[GP1:91,2] = PR[GP1:90,2] + 26.428;
   1:L PR[91] 10mm/sec CNT100;
   1:  PR[GP1:91,1] = PR[GP1:90,1] + -58.041;
   1:  PR[GP1:91,2] = PR[GP1:90,2] + 24.107;
   1:L PR[91] 10mm/sec CNT100;
   1:  PR[GP1:91,1] = PR[GP1:90,1] + -58.509;
   1:  PR[GP1:91,2] = PR[GP1:90,2] + 23.615;
   1:L PR[91] 10mm/sec CNT100;
   1:  PR[GP1:91,1] = PR[GP1:90,1] + -62.178;
   1:  PR[GP1:91,2] = PR[GP1:90,2] + 18.853;
   1:L PR[91] 10mm/sec CNT100;
   1:  PR[GP1:91,1] = PR[GP1:90,1] + -65.595;
   1:  PR[GP1:91,2] = PR[GP1:90,2] + 12.067;
   1:L PR[91] 10mm/sec CNT100;
   1:  PR[GP1:91,1] = PR[GP1:90,1] + -66.956;
   1:  PR[GP1:91,2] = PR[GP1:90,2] + 7.442;
   1:L PR[91] 10mm/sec CNT100;
   1:  PR[GP1:91,1] = PR[GP1:90,1] + -67.395;
   1:  PR[GP1:91,2] = PR[GP1:90,2] + 4.631;
   1:L PR[91] 10mm/sec CNT100;
   1:  PR[GP1:91,1] = PR[GP1:90,1] + -67.809;
   1:  PR[GP1:91,2] = PR[GP1:90,2] + 0.016;
   1:L PR[91] 10mm/sec CNT100;
   1:  PR[GP1:91,1] = PR[GP1:90,1] + -67.363;
   1:  PR[GP1:91,2] = PR[GP1:90,2] + -2.813;
   1:L PR[91] 10mm/sec CNT100;
   1:  PR[GP1:91,1] = PR[GP1:90,1] + -66.951;
   1:  PR[GP1:91,2] = PR[GP1:90,2] + -7.470;
   1:L PR[91] 10mm/sec CNT100;
   1:  PR[GP1:91,1] = PR[GP1:90,1] + -65.595;
   1:  PR[GP1:91,2] = PR[GP1:90,2] + -12.076;
   1:L PR[91] 10mm/sec CNT100;
   1:  PR[GP1:91,1] = PR[GP1:90,1] + -62.178;
   1:  PR[GP1:91,2] = PR[GP1:90,2] + -18.862;
   1:L PR[91] 10mm/sec CNT100;
   1:  PR[GP1:91,1] = PR[GP1:90,1] + -58.509;
   1:  PR[GP1:91,2] = PR[GP1:90,2] + -23.624;
   1:L PR[91] 10mm/sec CNT100;
   1:  PR[GP1:91,1] = PR[GP1:90,1] + -58.041;
   1:  PR[GP1:91,2] = PR[GP1:90,2] + -24.115;
   1:L PR[91] 10mm/sec CNT100;
   1:  PR[GP1:91,1] = PR[GP1:90,1] + -53.420;
   1:  PR[GP1:91,2] = PR[GP1:90,2] + -28.259;
   1:L PR[91] 10mm/sec CNT100;
   1:  PR[GP1:91,1] = PR[GP1:90,1] + -53.235;
   1:  PR[GP1:91,2] = PR[GP1:90,2] + -28.408;
   1:L PR[91] 10mm/sec CNT100;
   1:  PR[GP1:91,1] = PR[GP1:90,1] + -47.572;
   1:  PR[GP1:91,2] = PR[GP1:90,2] + -31.936;
   1:L PR[91] 10mm/sec CNT100;
   1:  PR[GP1:91,1] = PR[GP1:90,1] + -42.040;
   1:  PR[GP1:91,2] = PR[GP1:90,2] + -34.158;
   1:L PR[91] 10mm/sec CNT100;
   1:  PR[GP1:91,1] = PR[GP1:90,1] + -40.300;
   1:  PR[GP1:91,2] = PR[GP1:90,2] + -34.772;
   1:L PR[91] 10mm/sec CNT100;
   1:  PR[GP1:91,1] = PR[GP1:90,1] + -34.565;
   1:  PR[GP1:91,2] = PR[GP1:90,2] + -36.009;
   1:L PR[91] 10mm/sec CNT100;
   1:  PR[GP1:91,1] = PR[GP1:90,1] + -29.375;
   1:  PR[GP1:91,2] = PR[GP1:90,2] + -36.209;
   1:L PR[91] 10mm/sec CNT100;
   1:  PR[GP1:91,1] = PR[GP1:90,1] + -25.874;
   1:  PR[GP1:91,2] = PR[GP1:90,2] + -36.220;
   1:L PR[91] 10mm/sec CNT100;
   1:  PR[GP1:91,1] = PR[GP1:90,1] + -20.912;
   1:  PR[GP1:91,2] = PR[GP1:90,2] + -35.571;
   1:L PR[91] 10mm/sec CNT100;
   1:  PR[GP1:91,1] = PR[GP1:90,1] + -16.667;
   1:  PR[GP1:91,2] = PR[GP1:90,2] + -34.220;
   1:L PR[91] 10mm/sec CNT100;
   1:  PR[GP1:91,1] = PR[GP1:90,1] + -12.040;
   1:  PR[GP1:91,2] = PR[GP1:90,2] + -32.612;
   1:L PR[91] 10mm/sec CNT100;
   1:  PR[GP1:91,1] = PR[GP1:90,1] + -8.309;
   1:  PR[GP1:91,2] = PR[GP1:90,2] + -30.661;
   1:L PR[91] 10mm/sec CNT100;
   1:  PR[GP1:91,1] = PR[GP1:90,1] + -5.162;
   1:  PR[GP1:91,2] = PR[GP1:90,2] + -28.374;
   1:L PR[91] 10mm/sec CNT100;
   1:  PR[GP1:91,1] = PR[GP1:90,1] + -3.987;
   1:  PR[GP1:91,2] = PR[GP1:90,2] + -27.454;
   1:L PR[91] 10mm/sec CNT100;
   1:  PR[GP1:91,1] = PR[GP1:90,1] + -3.013;
   1:  PR[GP1:91,2] = PR[GP1:90,2] + -26.324;
   1:L PR[91] 10mm/sec CNT100;
   1:  PR[GP1:91,1] = PR[GP1:90,1] + 0.329;
   1:  PR[GP1:91,2] = PR[GP1:90,2] + -25.607;
   1:L PR[91] 10mm/sec CNT100;
   1:  PR[GP1:91,1] = PR[GP1:90,1] + 1.312;
   1:  PR[GP1:91,2] = PR[GP1:90,2] + -25.086;
   1:L PR[91] 10mm/sec CNT100;
   1:  PR[GP1:91,1] = PR[GP1:90,1] + 3.887;
   1:  PR[GP1:91,2] = PR[GP1:90,2] + -26.388;
   1:L PR[91] 10mm/sec CNT100;
   1:  PR[GP1:91,1] = PR[GP1:90,1] + 4.816;
   1:  PR[GP1:91,2] = PR[GP1:90,2] + -27.466;
   1:L PR[91] 10mm/sec CNT100;
   1:  PR[GP1:91,1] = PR[GP1:90,1] + 5.985;
   1:  PR[GP1:91,2] = PR[GP1:90,2] + -28.381;
   1:L PR[91] 10mm/sec CNT100;
   1:  PR[GP1:91,1] = PR[GP1:90,1] + 9.140;
   1:  PR[GP1:91,2] = PR[GP1:90,2] + -30.672;
   1:L PR[91] 10mm/sec CNT100;
   1:  PR[GP1:91,1] = PR[GP1:90,1] + 12.841;
   1:  PR[GP1:91,2] = PR[GP1:90,2] + -32.604;
   1:L PR[91] 10mm/sec CNT100;
   1:  PR[GP1:91,1] = PR[GP1:90,1] + 17.427;
   1:  PR[GP1:91,2] = PR[GP1:90,2] + -34.077;
   1:L PR[91] 10mm/sec CNT100;
   1:  PR[GP1:91,1] = PR[GP1:90,1] + 21.735;
   1:  PR[GP1:91,2] = PR[GP1:90,2] + -35.569;
   1:L PR[91] 10mm/sec CNT100;
   1:  PR[GP1:91,1] = PR[GP1:90,1] + 26.674;
   1:  PR[GP1:91,2] = PR[GP1:90,2] + -36.218;
   1:L PR[91] 10mm/sec CNT100;
   1:  PR[GP1:91,1] = PR[GP1:90,1] + 32.432;
   1:  PR[GP1:91,2] = PR[GP1:90,2] + -36.025;
   1:L PR[91] 10mm/sec CNT100;
   1:  PR[GP1:91,1] = PR[GP1:90,1] + 35.360;
   1:  PR[GP1:91,2] = PR[GP1:90,2] + -36.012;
   1:L PR[91] 10mm/sec CNT100;
   1:  PR[GP1:91,1] = PR[GP1:90,1] + 41.065;
   1:  PR[GP1:91,2] = PR[GP1:90,2] + -34.784;
   1:L PR[91] 10mm/sec CNT100;
   1:  PR[GP1:91,1] = PR[GP1:90,1] + 47.317;
   1:  PR[GP1:91,2] = PR[GP1:90,2] + -32.321;
   1:L PR[91] 10mm/sec CNT100;
   1:  PR[GP1:91,1] = PR[GP1:90,1] + 48.370;
   1:  PR[GP1:91,2] = PR[GP1:90,2] + -31.948;
   1:L PR[91] 10mm/sec CNT100;
   1:  PR[GP1:91,1] = PR[GP1:90,1] + 53.976;
   1:  PR[GP1:91,2] = PR[GP1:90,2] + -28.473;
   1:L PR[91] 10mm/sec CNT100;
   1:  PR[GP1:91,1] = PR[GP1:90,1] + 58.790;
   1:  PR[GP1:91,2] = PR[GP1:90,2] + -24.189;
   1:L PR[91] 10mm/sec CNT100;
   1:  PR[GP1:91,1] = PR[GP1:90,1] + 59.244;
   1:  PR[GP1:91,2] = PR[GP1:90,2] + -23.711;
   1:L PR[91] 10mm/sec CNT100;
   1:  PR[GP1:91,1] = PR[GP1:90,1] + 62.967;
   1:  PR[GP1:91,2] = PR[GP1:90,2] + -18.892;
   1:L PR[91] 10mm/sec CNT100;
   1:  PR[GP1:91,1] = PR[GP1:90,1] + 66.394;
   1:  PR[GP1:91,2] = PR[GP1:90,2] + -12.151;
   1:L PR[91] 10mm/sec CNT100;
   1:  PR[GP1:91,1] = PR[GP1:90,1] + 67.756;
   1:  PR[GP1:91,2] = PR[GP1:90,2] + -7.588;
   1:L PR[91] 10mm/sec CNT100;
   1:  PR[GP1:91,1] = PR[GP1:90,1] + 68.194;
   1:  PR[GP1:91,2] = PR[GP1:90,2] + -4.772;
   1:L PR[91] 10mm/sec CNT100;
   1:  PR[GP1:91,1] = PR[GP1:90,1] + 68.630;
   1:  PR[GP1:91,2] = PR[GP1:90,2] + -0.024;
   1:L PR[91] 10mm/sec CNT100;
   1:  PR[GP1:91,1] = PR[GP1:90,1] + 68.183;
   1:  PR[GP1:91,2] = PR[GP1:90,2] + 2.812;
   1:L PR[91] 10mm/sec CNT100;
   1:  PR[GP1:91,1] = PR[GP1:90,1] + 67.751;
   1:  PR[GP1:91,2] = PR[GP1:90,2] + 7.598;
   1:L PR[91] 10mm/sec CNT100;
   1:  PR[GP1:91,1] = PR[GP1:90,1] + 66.394;
   1:  PR[GP1:91,2] = PR[GP1:90,2] + 12.144;
   1:L PR[91] 10mm/sec CNT100;
   1:  PR[GP1:91,1] = PR[GP1:90,1] + 65.373;
   1:  PR[GP1:91,2] = PR[GP1:90,2] + 14.177;
   1:L PR[91] 10mm/sec CNT100;
   1:  PR[GP1:91,1] = PR[GP1:90,1] + 62.968;
   1:  PR[GP1:91,2] = PR[GP1:90,2] + 18.882;
   1:L PR[91] 10mm/sec CNT100;
   1:  PR[GP1:91,1] = PR[GP1:90,1] + 59.244;
   1:  PR[GP1:91,2] = PR[GP1:90,2] + 23.702;
   1:L PR[91] 10mm/sec CNT100;
   1:  PR[GP1:91,1] = PR[GP1:90,1] + 58.790;
   1:  PR[GP1:91,2] = PR[GP1:90,2] + 24.181;
   1:L PR[91] 10mm/sec CNT100;
   1:  PR[GP1:91,1] = PR[GP1:90,1] + 54.180;
   1:  PR[GP1:91,2] = PR[GP1:90,2] + 28.302;
   1:L PR[91] 10mm/sec CNT100;
   1:  PR[GP1:91,1] = PR[GP1:90,1] + 53.988;
   1:  PR[GP1:91,2] = PR[GP1:90,2] + 28.456;
   1:L PR[91] 10mm/sec CNT100;
   1:  PR[GP1:91,1] = PR[GP1:90,1] + 48.361;
   1:  PR[GP1:91,2] = PR[GP1:90,2] + 31.945;
   1:L PR[91] 10mm/sec CNT100;
   1:  PR[GP1:91,1] = PR[GP1:90,1] + 42.823;
   1:  PR[GP1:91,2] = PR[GP1:90,2] + 34.157;
   1:L PR[91] 10mm/sec CNT100;
   1:  PR[GP1:91,1] = PR[GP1:90,1] + 41.078;
   1:  PR[GP1:91,2] = PR[GP1:90,2] + 34.772;
   1:L PR[91] 10mm/sec CNT100;
   1:  PR[GP1:91,1] = PR[GP1:90,1] + 35.354;
   1:  PR[GP1:91,2] = PR[GP1:90,2] + 36.005;
   1:L PR[91] 10mm/sec CNT100;
   1:  PR[GP1:91,1] = PR[GP1:90,1] + 30.189;
   1:  PR[GP1:91,2] = PR[GP1:90,2] + 36.199;
   1:L PR[91] 10mm/sec CNT100;
   1:  PR[GP1:91,1] = PR[GP1:90,1] + 26.689;
   1:  PR[GP1:91,2] = PR[GP1:90,2] + 36.212;
   1:L PR[91] 10mm/sec CNT100;
   1:  PR[GP1:91,1] = PR[GP1:90,1] + 21.734;
   1:  PR[GP1:91,2] = PR[GP1:90,2] + 35.560;
   1:L PR[91] 10mm/sec CNT100;
   1:  PR[GP1:91,1] = PR[GP1:90,1] + 17.485;
   1:  PR[GP1:91,2] = PR[GP1:90,2] + 34.208;
   1:L PR[91] 10mm/sec CNT100;
   1:  PR[GP1:91,1] = PR[GP1:90,1] + 12.855;
   1:  PR[GP1:91,2] = PR[GP1:90,2] + 32.603;
   1:L PR[91] 10mm/sec CNT100;
   1:  PR[GP1:91,1] = PR[GP1:90,1] + 9.141;
   1:  PR[GP1:91,2] = PR[GP1:90,2] + 30.665;
   1:L PR[91] 10mm/sec CNT100;
   1:  PR[GP1:91,1] = PR[GP1:90,1] + 6.856;
   1:  PR[GP1:91,2] = PR[GP1:90,2] + 29.051;
   1:L PR[91] 10mm/sec CNT100;
   1:  PR[GP1:91,1] = PR[GP1:90,1] + 5.198;
   1:  PR[GP1:91,2] = PR[GP1:90,2] + 27.753;
   1:L PR[91] 10mm/sec CNT100;
   1:  PR[GP1:91,1] = PR[GP1:90,1] + 3.871;
   1:  PR[GP1:91,2] = PR[GP1:90,2] + 26.209;
   1:L PR[91] 10mm/sec CNT100;
   1:  PR[GP1:91,1] = PR[GP1:90,1] + 2.377;
   1:  PR[GP1:91,2] = PR[GP1:90,2] + 25.619;
   1:L PR[91] 10mm/sec CNT100;
   1:  PR[GP1:91,1] = PR[GP1:90,1] + 1.426;
   1:  PR[GP1:91,2] = PR[GP1:90,2] + 25.133;
   1:L PR[91] 10mm/sec CNT100;
   1:  PR[GP1:91,1] = PR[GP1:90,1] + -1.894;
   1:  PR[GP1:91,2] = PR[GP1:90,2] + 26.291;
   1:  PR[GP1:91,3] = PR[GP1:90,3] + 53.200;
   1:L PR[91] 10mm/sec CNT100;
   1:  PR[GP1:91,1] = PR[GP1:90,1] + -3.006;
   1:  PR[GP1:91,2] = PR[GP1:90,2] + 26.856;
   1:L PR[91] 10mm/sec CNT100;
   1:  PR[GP1:91,1] = PR[GP1:90,1] + -4.026;
   1:  PR[GP1:91,2] = PR[GP1:90,2] + 28.042;
   1:L PR[91] 10mm/sec CNT100;
   1:  PR[GP1:91,1] = PR[GP1:90,1] + -5.313;
   1:  PR[GP1:91,2] = PR[GP1:90,2] + 29.050;
   1:L PR[91] 10mm/sec CNT100;
   1:  PR[GP1:91,1] = PR[GP1:90,1] + -7.851;
   1:  PR[GP1:91,2] = PR[GP1:90,2] + 30.843;
   1:L PR[91] 10mm/sec CNT100;
   1:  PR[GP1:91,1] = PR[GP1:90,1] + -11.296;
   1:  PR[GP1:91,2] = PR[GP1:90,2] + 32.646;
   1:L PR[91] 10mm/sec CNT100;
   1:  PR[GP1:91,1] = PR[GP1:90,1] + -15.532;
   1:  PR[GP1:91,2] = PR[GP1:90,2] + 34.006;
   1:L PR[91] 10mm/sec CNT100;
   1:  PR[GP1:91,1] = PR[GP1:90,1] + -20.494;
   1:  PR[GP1:91,2] = PR[GP1:90,2] + 35.722;
   1:L PR[91] 10mm/sec CNT100;
   1:  PR[GP1:91,1] = PR[GP1:90,1] + -25.104;
   1:  PR[GP1:91,2] = PR[GP1:90,2] + 36.324;
   1:L PR[91] 10mm/sec CNT100;
   1:  PR[GP1:91,1] = PR[GP1:90,1] + -30.504;
   1:  PR[GP1:91,2] = PR[GP1:90,2] + 36.139;
   1:L PR[91] 10mm/sec CNT100;
   1:  PR[GP1:91,1] = PR[GP1:90,1] + -34.169;
   1:  PR[GP1:91,2] = PR[GP1:90,2] + 36.120;
   1:L PR[91] 10mm/sec CNT100;
   1:  PR[GP1:91,1] = PR[GP1:90,1] + -39.538;
   1:  PR[GP1:91,2] = PR[GP1:90,2] + 34.962;
   1:L PR[91] 10mm/sec CNT100;
   1:  PR[GP1:91,1] = PR[GP1:90,1] + -45.410;
   1:  PR[GP1:91,2] = PR[GP1:90,2] + 32.637;
   1:L PR[91] 10mm/sec CNT100;
   1:  PR[GP1:91,1] = PR[GP1:90,1] + -47.183;
   1:  PR[GP1:91,2] = PR[GP1:90,2] + 32.008;
   1:L PR[91] 10mm/sec CNT100;
   1:  PR[GP1:91,1] = PR[GP1:90,1] + -52.515;
   1:  PR[GP1:91,2] = PR[GP1:90,2] + 28.686;
   1:L PR[91] 10mm/sec CNT100;
   1:  PR[GP1:91,1] = PR[GP1:90,1] + -57.685;
   1:  PR[GP1:91,2] = PR[GP1:90,2] + 24.095;
   1:L PR[91] 10mm/sec CNT100;
   1:  PR[GP1:91,1] = PR[GP1:90,1] + -57.913;
   1:  PR[GP1:91,2] = PR[GP1:90,2] + 23.910;
   1:L PR[91] 10mm/sec CNT100;
   1:  PR[GP1:91,1] = PR[GP1:90,1] + -61.906;
   1:  PR[GP1:91,2] = PR[GP1:90,2] + 18.720;
   1:L PR[91] 10mm/sec CNT100;
   1:  PR[GP1:91,1] = PR[GP1:90,1] + -65.122;
   1:  PR[GP1:91,2] = PR[GP1:90,2] + 12.342;
   1:L PR[91] 10mm/sec CNT100;
   1:  PR[GP1:91,1] = PR[GP1:90,1] + -66.702;
   1:  PR[GP1:91,2] = PR[GP1:90,2] + 6.975;
   1:L PR[91] 10mm/sec CNT100;
   1:  PR[GP1:91,1] = PR[GP1:90,1] + -66.944;
   1:  PR[GP1:91,2] = PR[GP1:90,2] + 5.423;
   1:L PR[91] 10mm/sec CNT100;
   1:  PR[GP1:91,1] = PR[GP1:90,1] + -67.430;
   1:  PR[GP1:91,2] = PR[GP1:90,2] + 0.016;
   1:L PR[91] 10mm/sec CNT100;
   1:  PR[GP1:91,1] = PR[GP1:90,1] + -67.174;
   1:  PR[GP1:91,2] = PR[GP1:90,2] + -1.607;
   1:L PR[91] 10mm/sec CNT100;
   1:  PR[GP1:91,1] = PR[GP1:90,1] + -66.697;
   1:  PR[GP1:91,2] = PR[GP1:90,2] + -7.003;
   1:L PR[91] 10mm/sec CNT100;
   1:  PR[GP1:91,1] = PR[GP1:90,1] + -65.122;
   1:  PR[GP1:91,2] = PR[GP1:90,2] + -12.351;
   1:L PR[91] 10mm/sec CNT100;
   1:  PR[GP1:91,1] = PR[GP1:90,1] + -61.906;
   1:  PR[GP1:91,2] = PR[GP1:90,2] + -18.729;
   1:L PR[91] 10mm/sec CNT100;
   1:  PR[GP1:91,1] = PR[GP1:90,1] + -57.904;
   1:  PR[GP1:91,2] = PR[GP1:90,2] + -23.932;
   1:L PR[91] 10mm/sec CNT100;
   1:  PR[GP1:91,1] = PR[GP1:90,1] + -53.267;
   1:  PR[GP1:91,2] = PR[GP1:90,2] + -28.091;
   1:L PR[91] 10mm/sec CNT100;
   1:  PR[GP1:91,1] = PR[GP1:90,1] + -52.526;
   1:  PR[GP1:91,2] = PR[GP1:90,2] + -28.688;
   1:L PR[91] 10mm/sec CNT100;
   1:  PR[GP1:91,1] = PR[GP1:90,1] + -47.171;
   1:  PR[GP1:91,2] = PR[GP1:90,2] + -32.024;
   1:L PR[91] 10mm/sec CNT100;
   1:  PR[GP1:91,1] = PR[GP1:90,1] + -41.940;
   1:  PR[GP1:91,2] = PR[GP1:90,2] + -34.124;
   1:L PR[91] 10mm/sec CNT100;
   1:  PR[GP1:91,1] = PR[GP1:90,1] + -39.546;
   1:  PR[GP1:91,2] = PR[GP1:90,2] + -34.969;
   1:L PR[91] 10mm/sec CNT100;
   1:  PR[GP1:91,1] = PR[GP1:90,1] + -34.155;
   1:  PR[GP1:91,2] = PR[GP1:90,2] + -36.132;
   1:L PR[91] 10mm/sec CNT100;
   1:  PR[GP1:91,1] = PR[GP1:90,1] + -29.275;
   1:  PR[GP1:91,2] = PR[GP1:90,2] + -36.320;
   1:L PR[91] 10mm/sec CNT100;
   1:  PR[GP1:91,1] = PR[GP1:90,1] + -25.107;
   1:  PR[GP1:91,2] = PR[GP1:90,2] + -36.333;
   1:L PR[91] 10mm/sec CNT100;
   1:  PR[GP1:91,1] = PR[GP1:90,1] + -20.478;
   1:  PR[GP1:91,2] = PR[GP1:90,2] + -35.728;
   1:L PR[91] 10mm/sec CNT100;
   1:  PR[GP1:91,1] = PR[GP1:90,1] + -16.518;
   1:  PR[GP1:91,2] = PR[GP1:90,2] + -34.468;
   1:L PR[91] 10mm/sec CNT100;
   1:  PR[GP1:91,1] = PR[GP1:90,1] + -11.294;
   1:  PR[GP1:91,2] = PR[GP1:90,2] + -32.653;
   1:L PR[91] 10mm/sec CNT100;
   1:  PR[GP1:91,1] = PR[GP1:90,1] + -7.849;
   1:  PR[GP1:91,2] = PR[GP1:90,2] + -30.851;
   1:L PR[91] 10mm/sec CNT100;
   1:  PR[GP1:91,1] = PR[GP1:90,1] + -4.346;
   1:  PR[GP1:91,2] = PR[GP1:90,2] + -28.305;
   1:L PR[91] 10mm/sec CNT100;
   1:  PR[GP1:91,1] = PR[GP1:90,1] + -3.609;
   1:  PR[GP1:91,2] = PR[GP1:90,2] + -27.728;
   1:L PR[91] 10mm/sec CNT100;
   1:  PR[GP1:91,1] = PR[GP1:90,1] + -2.949;
   1:  PR[GP1:91,2] = PR[GP1:90,2] + -26.963;
   1:L PR[91] 10mm/sec CNT100;
   1:  PR[GP1:91,1] = PR[GP1:90,1] + 0.693;
   1:  PR[GP1:91,2] = PR[GP1:90,2] + -26.181;
   1:L PR[91] 10mm/sec CNT100;
   1:  PR[GP1:91,1] = PR[GP1:90,1] + 1.402;
   1:  PR[GP1:91,2] = PR[GP1:90,2] + -25.805;
   1:L PR[91] 10mm/sec CNT100;
   1:  PR[GP1:91,1] = PR[GP1:90,1] + 3.822;
   1:  PR[GP1:91,2] = PR[GP1:90,2] + -27.027;
   1:L PR[91] 10mm/sec CNT100;
   1:  PR[GP1:91,1] = PR[GP1:90,1] + 4.434;
   1:  PR[GP1:91,2] = PR[GP1:90,2] + -27.737;
   1:L PR[91] 10mm/sec CNT100;
   1:  PR[GP1:91,1] = PR[GP1:90,1] + 5.167;
   1:  PR[GP1:91,2] = PR[GP1:90,2] + -28.310;
   1:L PR[91] 10mm/sec CNT100;
   1:  PR[GP1:91,1] = PR[GP1:90,1] + 8.678;
   1:  PR[GP1:91,2] = PR[GP1:90,2] + -30.862;
   1:L PR[91] 10mm/sec CNT100;
   1:  PR[GP1:91,1] = PR[GP1:90,1] + 12.095;
   1:  PR[GP1:91,2] = PR[GP1:90,2] + -32.645;
   1:L PR[91] 10mm/sec CNT100;
   1:  PR[GP1:91,1] = PR[GP1:90,1] + 16.333;
   1:  PR[GP1:91,2] = PR[GP1:90,2] + -34.006;
   1:L PR[91] 10mm/sec CNT100;
   1:  PR[GP1:91,1] = PR[GP1:90,1] + 21.302;
   1:  PR[GP1:91,2] = PR[GP1:90,2] + -35.726;
   1:L PR[91] 10mm/sec CNT100;
   1:  PR[GP1:91,1] = PR[GP1:90,1] + 25.907;
   1:  PR[GP1:91,2] = PR[GP1:90,2] + -36.332;
   1:L PR[91] 10mm/sec CNT100;
   1:  PR[GP1:91,1] = PR[GP1:90,1] + 31.281;
   1:  PR[GP1:91,2] = PR[GP1:90,2] + -36.151;
   1:L PR[91] 10mm/sec CNT100;
   1:  PR[GP1:91,1] = PR[GP1:90,1] + 34.952;
   1:  PR[GP1:91,2] = PR[GP1:90,2] + -36.135;
   1:L PR[91] 10mm/sec CNT100;
   1:  PR[GP1:91,1] = PR[GP1:90,1] + 40.313;
   1:  PR[GP1:91,2] = PR[GP1:90,2] + -34.981;
   1:L PR[91] 10mm/sec CNT100;
   1:  PR[GP1:91,1] = PR[GP1:90,1] + 46.194;
   1:  PR[GP1:91,2] = PR[GP1:90,2] + -32.665;
   1:L PR[91] 10mm/sec CNT100;
   1:  PR[GP1:91,1] = PR[GP1:90,1] + 47.972;
   1:  PR[GP1:91,2] = PR[GP1:90,2] + -32.034;
   1:L PR[91] 10mm/sec CNT100;
   1:  PR[GP1:91,1] = PR[GP1:90,1] + 53.271;
   1:  PR[GP1:91,2] = PR[GP1:90,2] + -28.750;
   1:L PR[91] 10mm/sec CNT100;
   1:  PR[GP1:91,1] = PR[GP1:90,1] + 58.413;
   1:  PR[GP1:91,2] = PR[GP1:90,2] + -24.196;
   1:L PR[91] 10mm/sec CNT100;
   1:  PR[GP1:91,1] = PR[GP1:90,1] + 58.651;
   1:  PR[GP1:91,2] = PR[GP1:90,2] + -24.004;
   1:L PR[91] 10mm/sec CNT100;
   1:  PR[GP1:91,1] = PR[GP1:90,1] + 62.691;
   1:  PR[GP1:91,2] = PR[GP1:90,2] + -18.765;
   1:L PR[91] 10mm/sec CNT100;
   1:  PR[GP1:91,1] = PR[GP1:90,1] + 65.918;
   1:  PR[GP1:91,2] = PR[GP1:90,2] + -12.434;
   1:L PR[91] 10mm/sec CNT100;
   1:  PR[GP1:91,1] = PR[GP1:90,1] + 67.499;
   1:  PR[GP1:91,2] = PR[GP1:90,2] + -7.138;
   1:L PR[91] 10mm/sec CNT100;
   1:  PR[GP1:91,1] = PR[GP1:90,1] + 67.740;
   1:  PR[GP1:91,2] = PR[GP1:90,2] + -5.588;
   1:L PR[91] 10mm/sec CNT100;
   1:  PR[GP1:91,1] = PR[GP1:90,1] + 68.251;
   1:  PR[GP1:91,2] = PR[GP1:90,2] + -0.024;
   1:L PR[91] 10mm/sec CNT100;
   1:  PR[GP1:91,1] = PR[GP1:90,1] + 67.995;
   1:  PR[GP1:91,2] = PR[GP1:90,2] + 1.603;
   1:L PR[91] 10mm/sec CNT100;
   1:  PR[GP1:91,1] = PR[GP1:90,1] + 67.493;
   1:  PR[GP1:91,2] = PR[GP1:90,2] + 7.148;
   1:L PR[91] 10mm/sec CNT100;
   1:  PR[GP1:91,1] = PR[GP1:90,1] + 65.918;
   1:  PR[GP1:91,2] = PR[GP1:90,2] + 12.425;
   1:L PR[91] 10mm/sec CNT100;
   1:  PR[GP1:91,1] = PR[GP1:90,1] + 62.691;
   1:  PR[GP1:91,2] = PR[GP1:90,2] + 18.756;
   1:L PR[91] 10mm/sec CNT100;
   1:  PR[GP1:91,1] = PR[GP1:90,1] + 58.642;
   1:  PR[GP1:91,2] = PR[GP1:90,2] + 24.007;
   1:L PR[91] 10mm/sec CNT100;
   1:  PR[GP1:91,1] = PR[GP1:90,1] + 54.030;
   1:  PR[GP1:91,2] = PR[GP1:90,2] + 28.130;
   1:L PR[91] 10mm/sec CNT100;
   1:  PR[GP1:91,1] = PR[GP1:90,1] + 53.283;
   1:  PR[GP1:91,2] = PR[GP1:90,2] + 28.733;
   1:L PR[91] 10mm/sec CNT100;
   1:  PR[GP1:91,1] = PR[GP1:90,1] + 47.963;
   1:  PR[GP1:91,2] = PR[GP1:90,2] + 32.031;
   1:L PR[91] 10mm/sec CNT100;
   1:  PR[GP1:91,1] = PR[GP1:90,1] + 42.725;
   1:  PR[GP1:91,2] = PR[GP1:90,2] + 34.123;
   1:L PR[91] 10mm/sec CNT100;
   1:  PR[GP1:91,1] = PR[GP1:90,1] + 40.327;
   1:  PR[GP1:91,2] = PR[GP1:90,2] + 34.969;
   1:L PR[91] 10mm/sec CNT100;
   1:  PR[GP1:91,1] = PR[GP1:90,1] + 34.946;
   1:  PR[GP1:91,2] = PR[GP1:90,2] + 36.128;
   1:L PR[91] 10mm/sec CNT100;
   1:  PR[GP1:91,1] = PR[GP1:90,1] + 30.090;
   1:  PR[GP1:91,2] = PR[GP1:90,2] + 36.311;
   1:L PR[91] 10mm/sec CNT100;
   1:  PR[GP1:91,1] = PR[GP1:90,1] + 25.923;
   1:  PR[GP1:91,2] = PR[GP1:90,2] + 36.325;
   1:L PR[91] 10mm/sec CNT100;
   1:  PR[GP1:91,1] = PR[GP1:90,1] + 21.302;
   1:  PR[GP1:91,2] = PR[GP1:90,2] + 35.718;
   1:L PR[91] 10mm/sec CNT100;
   1:  PR[GP1:91,1] = PR[GP1:90,1] + 17.337;
   1:  PR[GP1:91,2] = PR[GP1:90,2] + 34.456;
   1:L PR[91] 10mm/sec CNT100;
   1:  PR[GP1:91,1] = PR[GP1:90,1] + 12.110;
   1:  PR[GP1:91,2] = PR[GP1:90,2] + 32.644;
   1:L PR[91] 10mm/sec CNT100;
   1:  PR[GP1:91,1] = PR[GP1:90,1] + 8.680;
   1:  PR[GP1:91,2] = PR[GP1:90,2] + 30.854;
   1:L PR[91] 10mm/sec CNT100;
   1:  PR[GP1:91,1] = PR[GP1:90,1] + 6.135;
   1:  PR[GP1:91,2] = PR[GP1:90,2] + 29.057;
   1:L PR[91] 10mm/sec CNT100;
   1:  PR[GP1:91,1] = PR[GP1:90,1] + 4.854;
   1:  PR[GP1:91,2] = PR[GP1:90,2] + 28.054;
   1:L PR[91] 10mm/sec CNT100;
   1:  PR[GP1:91,1] = PR[GP1:90,1] + 3.806;
   1:  PR[GP1:91,2] = PR[GP1:90,2] + 26.834;
   1:L PR[91] 10mm/sec CNT100;
   1:  PR[GP1:91,1] = PR[GP1:90,1] + 2.184;
   1:  PR[GP1:91,2] = PR[GP1:90,2] + 26.194;
   1:L PR[91] 10mm/sec CNT100;
   1:  PR[GP1:91,1] = PR[GP1:90,1] + 1.516;
   1:  PR[GP1:91,2] = PR[GP1:90,2] + 25.852;
   1:L PR[91] 10mm/sec CNT100;
   1:  PR[GP1:91,1] = PR[GP1:90,1] + -2.088;
   1:  PR[GP1:91,2] = PR[GP1:90,2] + 27.046;
   1:  PR[GP1:91,3] = PR[GP1:90,3] + 54.530;
   1:L PR[91] 10mm/sec CNT100;
   1:  PR[GP1:91,1] = PR[GP1:90,1] + -2.942;
   1:  PR[GP1:91,2] = PR[GP1:90,2] + 27.481;
   1:L PR[91] 10mm/sec CNT100;
   1:  PR[GP1:91,1] = PR[GP1:90,1] + -3.686;
   1:  PR[GP1:91,2] = PR[GP1:90,2] + 28.346;
   1:L PR[91] 10mm/sec CNT100;
   1:  PR[GP1:91,1] = PR[GP1:90,1] + -4.595;
   1:  PR[GP1:91,2] = PR[GP1:90,2] + 29.057;
   1:L PR[91] 10mm/sec CNT100;
   1:  PR[GP1:91,1] = PR[GP1:90,1] + -7.392;
   1:  PR[GP1:91,2] = PR[GP1:90,2] + 31.034;
   1:L PR[91] 10mm/sec CNT100;
   1:  PR[GP1:91,1] = PR[GP1:90,1] + -10.551;
   1:  PR[GP1:91,2] = PR[GP1:90,2] + 32.687;
   1:L PR[91] 10mm/sec CNT100;
   1:  PR[GP1:91,1] = PR[GP1:90,1] + -14.440;
   1:  PR[GP1:91,2] = PR[GP1:90,2] + 33.936;
   1:L PR[91] 10mm/sec CNT100;
   1:  PR[GP1:91,1] = PR[GP1:90,1] + -20.061;
   1:  PR[GP1:91,2] = PR[GP1:90,2] + 35.879;
   1:L PR[91] 10mm/sec CNT100;
   1:  PR[GP1:91,1] = PR[GP1:90,1] + -24.338;
   1:  PR[GP1:91,2] = PR[GP1:90,2] + 36.438;
   1:L PR[91] 10mm/sec CNT100;
   1:  PR[GP1:91,1] = PR[GP1:90,1] + -29.353;
   1:  PR[GP1:91,2] = PR[GP1:90,2] + 36.266;
   1:L PR[91] 10mm/sec CNT100;
   1:  PR[GP1:91,1] = PR[GP1:90,1] + -33.760;
   1:  PR[GP1:91,2] = PR[GP1:90,2] + 36.244;
   1:L PR[91] 10mm/sec CNT100;
   1:  PR[GP1:91,1] = PR[GP1:90,1] + -38.785;
   1:  PR[GP1:91,2] = PR[GP1:90,2] + 35.160;
   1:L PR[91] 10mm/sec CNT100;
   1:  PR[GP1:91,1] = PR[GP1:90,1] + -44.286;
   1:  PR[GP1:91,2] = PR[GP1:90,2] + 32.982;
   1:L PR[91] 10mm/sec CNT100;
   1:  PR[GP1:91,1] = PR[GP1:90,1] + -46.783;
   1:  PR[GP1:91,2] = PR[GP1:90,2] + 32.095;
   1:L PR[91] 10mm/sec CNT100;
   1:  PR[GP1:91,1] = PR[GP1:90,1] + -51.806;
   1:  PR[GP1:91,2] = PR[GP1:90,2] + 28.966;
   1:L PR[91] 10mm/sec CNT100;
   1:  PR[GP1:91,1] = PR[GP1:90,1] + -56.681;
   1:  PR[GP1:91,2] = PR[GP1:90,2] + 24.637;
   1:L PR[91] 10mm/sec CNT100;
   1:  PR[GP1:91,1] = PR[GP1:90,1] + -57.513;
   1:  PR[GP1:91,2] = PR[GP1:90,2] + 23.963;
   1:L PR[91] 10mm/sec CNT100;
   1:  PR[GP1:91,1] = PR[GP1:90,1] + -61.402;
   1:  PR[GP1:91,2] = PR[GP1:90,2] + 18.902;
   1:L PR[91] 10mm/sec CNT100;
   1:  PR[GP1:91,1] = PR[GP1:90,1] + -64.655;
   1:  PR[GP1:91,2] = PR[GP1:90,2] + 12.597;
   1:L PR[91] 10mm/sec CNT100;
   1:  PR[GP1:91,1] = PR[GP1:90,1] + -66.448;
   1:  PR[GP1:91,2] = PR[GP1:90,2] + 6.508;
   1:L PR[91] 10mm/sec CNT100;
   1:  PR[GP1:91,1] = PR[GP1:90,1] + -66.494;
   1:  PR[GP1:91,2] = PR[GP1:90,2] + 6.216;
   1:L PR[91] 10mm/sec CNT100;
   1:  PR[GP1:91,1] = PR[GP1:90,1] + -67.051;
   1:  PR[GP1:91,2] = PR[GP1:90,2] + 0.016;
   1:L PR[91] 10mm/sec CNT100;
   1:  PR[GP1:91,1] = PR[GP1:90,1] + -66.985;
   1:  PR[GP1:91,2] = PR[GP1:90,2] + -0.401;
   1:L PR[91] 10mm/sec CNT100;
   1:  PR[GP1:91,1] = PR[GP1:90,1] + -66.442;
   1:  PR[GP1:91,2] = PR[GP1:90,2] + -6.537;
   1:L PR[91] 10mm/sec CNT100;
   1:  PR[GP1:91,1] = PR[GP1:90,1] + -64.655;
   1:  PR[GP1:91,2] = PR[GP1:90,2] + -12.607;
   1:L PR[91] 10mm/sec CNT100;
   1:  PR[GP1:91,1] = PR[GP1:90,1] + -61.637;
   1:  PR[GP1:91,2] = PR[GP1:90,2] + -18.524;
   1:L PR[91] 10mm/sec CNT100;
   1:  PR[GP1:91,1] = PR[GP1:90,1] + -61.413;
   1:  PR[GP1:91,2] = PR[GP1:90,2] + -18.896;
   1:L PR[91] 10mm/sec CNT100;
   1:  PR[GP1:91,1] = PR[GP1:90,1] + -57.504;
   1:  PR[GP1:91,2] = PR[GP1:90,2] + -23.985;
   1:L PR[91] 10mm/sec CNT100;
   1:  PR[GP1:91,1] = PR[GP1:90,1] + -53.114;
   1:  PR[GP1:91,2] = PR[GP1:90,2] + -27.922;
   1:L PR[91] 10mm/sec CNT100;
   1:  PR[GP1:91,1] = PR[GP1:90,1] + -51.817;
   1:  PR[GP1:91,2] = PR[GP1:90,2] + -28.968;
   1:L PR[91] 10mm/sec CNT100;
   1:  PR[GP1:91,1] = PR[GP1:90,1] + -46.771;
   1:  PR[GP1:91,2] = PR[GP1:90,2] + -32.112;
   1:L PR[91] 10mm/sec CNT100;
   1:  PR[GP1:91,1] = PR[GP1:90,1] + -41.841;
   1:  PR[GP1:91,2] = PR[GP1:90,2] + -34.091;
   1:L PR[91] 10mm/sec CNT100;
   1:  PR[GP1:91,1] = PR[GP1:90,1] + -38.791;
   1:  PR[GP1:91,2] = PR[GP1:90,2] + -35.167;
   1:L PR[91] 10mm/sec CNT100;
   1:  PR[GP1:91,1] = PR[GP1:90,1] + -33.745;
   1:  PR[GP1:91,2] = PR[GP1:90,2] + -36.256;
   1:L PR[91] 10mm/sec CNT100;
   1:  PR[GP1:91,1] = PR[GP1:90,1] + -29.175;
   1:  PR[GP1:91,2] = PR[GP1:90,2] + -36.432;
   1:L PR[91] 10mm/sec CNT100;
   1:  PR[GP1:91,1] = PR[GP1:90,1] + -24.339;
   1:  PR[GP1:91,2] = PR[GP1:90,2] + -36.447;
   1:L PR[91] 10mm/sec CNT100;
   1:  PR[GP1:91,1] = PR[GP1:90,1] + -20.045;
   1:  PR[GP1:91,2] = PR[GP1:90,2] + -35.886;
   1:L PR[91] 10mm/sec CNT100;
   1:  PR[GP1:91,1] = PR[GP1:90,1] + -16.369;
   1:  PR[GP1:91,2] = PR[GP1:90,2] + -34.716;
   1:L PR[91] 10mm/sec CNT100;
   1:  PR[GP1:91,1] = PR[GP1:90,1] + -10.547;
   1:  PR[GP1:91,2] = PR[GP1:90,2] + -32.693;
   1:L PR[91] 10mm/sec CNT100;
   1:  PR[GP1:91,1] = PR[GP1:90,1] + -7.389;
   1:  PR[GP1:91,2] = PR[GP1:90,2] + -31.041;
   1:L PR[91] 10mm/sec CNT100;
   1:  PR[GP1:91,1] = PR[GP1:90,1] + -3.530;
   1:  PR[GP1:91,2] = PR[GP1:90,2] + -28.237;
   1:L PR[91] 10mm/sec CNT100;
   1:  PR[GP1:91,1] = PR[GP1:90,1] + -3.231;
   1:  PR[GP1:91,2] = PR[GP1:90,2] + -28.003;
   1:L PR[91] 10mm/sec CNT100;
   1:  PR[GP1:91,1] = PR[GP1:90,1] + -2.885;
   1:  PR[GP1:91,2] = PR[GP1:90,2] + -27.601;
   1:L PR[91] 10mm/sec CNT100;
   1:  PR[GP1:91,1] = PR[GP1:90,1] + 1.057;
   1:  PR[GP1:91,2] = PR[GP1:90,2] + -26.755;
   1:L PR[91] 10mm/sec CNT100;
   1:  PR[GP1:91,1] = PR[GP1:90,1] + 1.492;
   1:  PR[GP1:91,2] = PR[GP1:90,2] + -26.525;
   1:L PR[91] 10mm/sec CNT100;
   1:  PR[GP1:91,1] = PR[GP1:90,1] + 3.756;
   1:  PR[GP1:91,2] = PR[GP1:90,2] + -27.665;
   1:L PR[91] 10mm/sec CNT100;
   1:  PR[GP1:91,1] = PR[GP1:90,1] + 4.051;
   1:  PR[GP1:91,2] = PR[GP1:90,2] + -28.008;
   1:L PR[91] 10mm/sec CNT100;
   1:  PR[GP1:91,1] = PR[GP1:90,1] + 4.348;
   1:  PR[GP1:91,2] = PR[GP1:90,2] + -28.240;
   1:L PR[91] 10mm/sec CNT100;
   1:  PR[GP1:91,1] = PR[GP1:90,1] + 8.217;
   1:  PR[GP1:91,2] = PR[GP1:90,2] + -31.051;
   1:L PR[91] 10mm/sec CNT100;
   1:  PR[GP1:91,1] = PR[GP1:90,1] + 11.349;
   1:  PR[GP1:91,2] = PR[GP1:90,2] + -32.685;
   1:L PR[91] 10mm/sec CNT100;
   1:  PR[GP1:91,1] = PR[GP1:90,1] + 15.239;
   1:  PR[GP1:91,2] = PR[GP1:90,2] + -33.935;
   1:L PR[91] 10mm/sec CNT100;
   1:  PR[GP1:91,1] = PR[GP1:90,1] + 20.868;
   1:  PR[GP1:91,2] = PR[GP1:90,2] + -35.884;
   1:L PR[91] 10mm/sec CNT100;
   1:  PR[GP1:91,1] = PR[GP1:90,1] + 25.139;
   1:  PR[GP1:91,2] = PR[GP1:90,2] + -36.446;
   1:L PR[91] 10mm/sec CNT100;
   1:  PR[GP1:91,1] = PR[GP1:90,1] + 30.131;
   1:  PR[GP1:91,2] = PR[GP1:90,2] + -36.278;
   1:L PR[91] 10mm/sec CNT100;
   1:  PR[GP1:91,1] = PR[GP1:90,1] + 34.544;
   1:  PR[GP1:91,2] = PR[GP1:90,2] + -36.258;
   1:L PR[91] 10mm/sec CNT100;
   1:  PR[GP1:91,1] = PR[GP1:90,1] + 39.561;
   1:  PR[GP1:91,2] = PR[GP1:90,2] + -35.178;
   1:L PR[91] 10mm/sec CNT100;
   1:  PR[GP1:91,1] = PR[GP1:90,1] + 45.070;
   1:  PR[GP1:91,2] = PR[GP1:90,2] + -33.008;
   1:L PR[91] 10mm/sec CNT100;
   1:  PR[GP1:91,1] = PR[GP1:90,1] + 47.573;
   1:  PR[GP1:91,2] = PR[GP1:90,2] + -32.121;
   1:L PR[91] 10mm/sec CNT100;
   1:  PR[GP1:91,1] = PR[GP1:90,1] + 52.565;
   1:  PR[GP1:91,2] = PR[GP1:90,2] + -29.026;
   1:L PR[91] 10mm/sec CNT100;
   1:  PR[GP1:91,1] = PR[GP1:90,1] + 57.414;
   1:  PR[GP1:91,2] = PR[GP1:90,2] + -24.733;
   1:L PR[91] 10mm/sec CNT100;
   1:  PR[GP1:91,1] = PR[GP1:90,1] + 58.255;
   1:  PR[GP1:91,2] = PR[GP1:90,2] + -24.052;
   1:L PR[91] 10mm/sec CNT100;
   1:  PR[GP1:91,1] = PR[GP1:90,1] + 62.183;
   1:  PR[GP1:91,2] = PR[GP1:90,2] + -18.952;
   1:L PR[91] 10mm/sec CNT100;
   1:  PR[GP1:91,1] = PR[GP1:90,1] + 65.449;
   1:  PR[GP1:91,2] = PR[GP1:90,2] + -12.694;
   1:L PR[91] 10mm/sec CNT100;
   1:  PR[GP1:91,1] = PR[GP1:90,1] + 67.241;
   1:  PR[GP1:91,2] = PR[GP1:90,2] + -6.689;
   1:L PR[91] 10mm/sec CNT100;
   1:  PR[GP1:91,1] = PR[GP1:90,1] + 67.286;
   1:  PR[GP1:91,2] = PR[GP1:90,2] + -6.403;
   1:L PR[91] 10mm/sec CNT100;
   1:  PR[GP1:91,1] = PR[GP1:90,1] + 67.872;
   1:  PR[GP1:91,2] = PR[GP1:90,2] + -0.024;
   1:L PR[91] 10mm/sec CNT100;
   1:  PR[GP1:91,1] = PR[GP1:90,1] + 67.806;
   1:  PR[GP1:91,2] = PR[GP1:90,2] + 0.393;
   1:L PR[91] 10mm/sec CNT100;
   1:  PR[GP1:91,1] = PR[GP1:90,1] + 67.236;
   1:  PR[GP1:91,2] = PR[GP1:90,2] + 6.698;
   1:L PR[91] 10mm/sec CNT100;
   1:  PR[GP1:91,1] = PR[GP1:90,1] + 65.448;
   1:  PR[GP1:91,2] = PR[GP1:90,2] + 12.687;
   1:L PR[91] 10mm/sec CNT100;
   1:  PR[GP1:91,1] = PR[GP1:90,1] + 62.421;
   1:  PR[GP1:91,2] = PR[GP1:90,2] + 18.552;
   1:L PR[91] 10mm/sec CNT100;
   1:  PR[GP1:91,1] = PR[GP1:90,1] + 62.195;
   1:  PR[GP1:91,2] = PR[GP1:90,2] + 18.929;
   1:L PR[91] 10mm/sec CNT100;
   1:  PR[GP1:91,1] = PR[GP1:90,1] + 58.246;
   1:  PR[GP1:91,2] = PR[GP1:90,2] + 24.055;
   1:L PR[91] 10mm/sec CNT100;
   1:  PR[GP1:91,1] = PR[GP1:90,1] + 53.880;
   1:  PR[GP1:91,2] = PR[GP1:90,2] + 27.959;
   1:L PR[91] 10mm/sec CNT100;
   1:  PR[GP1:91,1] = PR[GP1:90,1] + 52.579;
   1:  PR[GP1:91,2] = PR[GP1:90,2] + 29.009;
   1:L PR[91] 10mm/sec CNT100;
   1:  PR[GP1:91,1] = PR[GP1:90,1] + 47.565;
   1:  PR[GP1:91,2] = PR[GP1:90,2] + 32.117;
   1:L PR[91] 10mm/sec CNT100;
   1:  PR[GP1:91,1] = PR[GP1:90,1] + 42.628;
   1:  PR[GP1:91,2] = PR[GP1:90,2] + 34.089;
   1:L PR[91] 10mm/sec CNT100;
   1:  PR[GP1:91,1] = PR[GP1:90,1] + 39.576;
   1:  PR[GP1:91,2] = PR[GP1:90,2] + 35.167;
   1:L PR[91] 10mm/sec CNT100;
   1:  PR[GP1:91,1] = PR[GP1:90,1] + 34.539;
   1:  PR[GP1:91,2] = PR[GP1:90,2] + 36.251;
   1:L PR[91] 10mm/sec CNT100;
   1:  PR[GP1:91,1] = PR[GP1:90,1] + 29.992;
   1:  PR[GP1:91,2] = PR[GP1:90,2] + 36.422;
   1:L PR[91] 10mm/sec CNT100;
   1:  PR[GP1:91,1] = PR[GP1:90,1] + 25.157;
   1:  PR[GP1:91,2] = PR[GP1:90,2] + 36.439;
   1:L PR[91] 10mm/sec CNT100;
   1:  PR[GP1:91,1] = PR[GP1:90,1] + 20.869;
   1:  PR[GP1:91,2] = PR[GP1:90,2] + 35.876;
   1:L PR[91] 10mm/sec CNT100;
   1:  PR[GP1:91,1] = PR[GP1:90,1] + 17.189;
   1:  PR[GP1:91,2] = PR[GP1:90,2] + 34.705;
   1:L PR[91] 10mm/sec CNT100;
   1:  PR[GP1:91,1] = PR[GP1:90,1] + 11.365;
   1:  PR[GP1:91,2] = PR[GP1:90,2] + 32.685;
   1:L PR[91] 10mm/sec CNT100;
   1:  PR[GP1:91,1] = PR[GP1:90,1] + 8.219;
   1:  PR[GP1:91,2] = PR[GP1:90,2] + 31.044;
   1:L PR[91] 10mm/sec CNT100;
   1:  PR[GP1:91,1] = PR[GP1:90,1] + 5.414;
   1:  PR[GP1:91,2] = PR[GP1:90,2] + 29.062;
   1:L PR[91] 10mm/sec CNT100;
   1:  PR[GP1:91,1] = PR[GP1:90,1] + 4.510;
   1:  PR[GP1:91,2] = PR[GP1:90,2] + 28.355;
   1:L PR[91] 10mm/sec CNT100;
   1:  PR[GP1:91,1] = PR[GP1:90,1] + 3.741;
   1:  PR[GP1:91,2] = PR[GP1:90,2] + 27.459;
   1:L PR[91] 10mm/sec CNT100;
   1:  PR[GP1:91,1] = PR[GP1:90,1] + 1.990;
   1:  PR[GP1:91,2] = PR[GP1:90,2] + 26.768;
   1:L PR[91] 10mm/sec CNT100;
   1:  PR[GP1:91,1] = PR[GP1:90,1] + 1.606;
   1:  PR[GP1:91,2] = PR[GP1:90,2] + 26.572;
   1:L PR[91] 10mm/sec CNT100;
   1:  PR[GP1:91,1] = PR[GP1:90,1] + 1.152;
   1:  PR[GP1:91,2] = PR[GP1:90,2] + 27.361;
   1:  PR[GP1:91,3] = PR[GP1:90,3] + 55.860;
   1:L PR[91] 10mm/sec CNT100;
   1:  PR[GP1:91,1] = PR[GP1:90,1] + -2.281;
   1:  PR[GP1:91,2] = PR[GP1:90,2] + 27.802;
   1:L PR[91] 10mm/sec CNT100;
   1:  PR[GP1:91,1] = PR[GP1:90,1] + -2.879;
   1:  PR[GP1:91,2] = PR[GP1:90,2] + 28.106;
   1:L PR[91] 10mm/sec CNT100;
   1:  PR[GP1:91,1] = PR[GP1:90,1] + -3.346;
   1:  PR[GP1:91,2] = PR[GP1:90,2] + 28.649;
   1:L PR[91] 10mm/sec CNT100;
   1:  PR[GP1:91,1] = PR[GP1:90,1] + -3.876;
   1:  PR[GP1:91,2] = PR[GP1:90,2] + 29.064;
   1:L PR[91] 10mm/sec CNT100;
   1:  PR[GP1:91,1] = PR[GP1:90,1] + -6.932;
   1:  PR[GP1:91,2] = PR[GP1:90,2] + 31.224;
   1:L PR[91] 10mm/sec CNT100;
   1:  PR[GP1:91,1] = PR[GP1:90,1] + -9.806;
   1:  PR[GP1:91,2] = PR[GP1:90,2] + 32.728;
   1:L PR[91] 10mm/sec CNT100;
   1:  PR[GP1:91,1] = PR[GP1:90,1] + -13.348;
   1:  PR[GP1:91,2] = PR[GP1:90,2] + 33.865;
   1:L PR[91] 10mm/sec CNT100;
   1:  PR[GP1:91,1] = PR[GP1:90,1] + -19.629;
   1:  PR[GP1:91,2] = PR[GP1:90,2] + 36.037;
   1:L PR[91] 10mm/sec CNT100;
   1:  PR[GP1:91,1] = PR[GP1:90,1] + -23.571;
   1:  PR[GP1:91,2] = PR[GP1:90,2] + 36.552;
   1:L PR[91] 10mm/sec CNT100;
   1:  PR[GP1:91,1] = PR[GP1:90,1] + -28.201;
   1:  PR[GP1:91,2] = PR[GP1:90,2] + 36.393;
   1:L PR[91] 10mm/sec CNT100;
   1:  PR[GP1:91,1] = PR[GP1:90,1] + -33.350;
   1:  PR[GP1:91,2] = PR[GP1:90,2] + 36.367;
   1:L PR[91] 10mm/sec CNT100;
   1:  PR[GP1:91,1] = PR[GP1:90,1] + -38.031;
   1:  PR[GP1:91,2] = PR[GP1:90,2] + 35.357;
   1:L PR[91] 10mm/sec CNT100;
   1:  PR[GP1:91,1] = PR[GP1:90,1] + -43.161;
   1:  PR[GP1:91,2] = PR[GP1:90,2] + 33.326;
   1:L PR[91] 10mm/sec CNT100;
   1:  PR[GP1:91,1] = PR[GP1:90,1] + -46.383;
   1:  PR[GP1:91,2] = PR[GP1:90,2] + 32.182;
   1:L PR[91] 10mm/sec CNT100;
   1:  PR[GP1:91,1] = PR[GP1:90,1] + -51.098;
   1:  PR[GP1:91,2] = PR[GP1:90,2] + 29.245;
   1:L PR[91] 10mm/sec CNT100;
   1:  PR[GP1:91,1] = PR[GP1:90,1] + -55.678;
   1:  PR[GP1:91,2] = PR[GP1:90,2] + 25.178;
   1:L PR[91] 10mm/sec CNT100;
   1:  PR[GP1:91,1] = PR[GP1:90,1] + -57.114;
   1:  PR[GP1:91,2] = PR[GP1:90,2] + 24.016;
   1:L PR[91] 10mm/sec CNT100;
   1:  PR[GP1:91,1] = PR[GP1:90,1] + -60.781;
   1:  PR[GP1:91,2] = PR[GP1:90,2] + 19.243;
   1:L PR[91] 10mm/sec CNT100;
   1:  PR[GP1:91,1] = PR[GP1:90,1] + -63.858;
   1:  PR[GP1:91,2] = PR[GP1:90,2] + 13.272;
   1:L PR[91] 10mm/sec CNT100;
   1:  PR[GP1:91,1] = PR[GP1:90,1] + -64.253;
   1:  PR[GP1:91,2] = PR[GP1:90,2] + 12.613;
   1:L PR[91] 10mm/sec CNT100;
   1:  PR[GP1:91,1] = PR[GP1:90,1] + -66.005;
   1:  PR[GP1:91,2] = PR[GP1:90,2] + 6.667;
   1:L PR[91] 10mm/sec CNT100;
   1:  PR[GP1:91,1] = PR[GP1:90,1] + -66.583;
   1:  PR[GP1:91,2] = PR[GP1:90,2] + 0.358;
   1:L PR[91] 10mm/sec CNT100;
   1:  PR[GP1:91,1] = PR[GP1:90,1] + -66.655;
   1:  PR[GP1:91,2] = PR[GP1:90,2] + -0.032;
   1:L PR[91] 10mm/sec CNT100;
   1:  PR[GP1:91,1] = PR[GP1:90,1] + -66.098;
   1:  PR[GP1:91,2] = PR[GP1:90,2] + -6.191;
   1:L PR[91] 10mm/sec CNT100;
   1:  PR[GP1:91,1] = PR[GP1:90,1] + -66.013;
   1:  PR[GP1:91,2] = PR[GP1:90,2] + -6.649;
   1:L PR[91] 10mm/sec CNT100;
   1:  PR[GP1:91,1] = PR[GP1:90,1] + -64.247;
   1:  PR[GP1:91,2] = PR[GP1:90,2] + -12.642;
   1:L PR[91] 10mm/sec CNT100;
   1:  PR[GP1:91,1] = PR[GP1:90,1] + -61.391;
   1:  PR[GP1:91,2] = PR[GP1:90,2] + -18.241;
   1:L PR[91] 10mm/sec CNT100;
   1:  PR[GP1:91,1] = PR[GP1:90,1] + -60.793;
   1:  PR[GP1:91,2] = PR[GP1:90,2] + -19.236;
   1:L PR[91] 10mm/sec CNT100;
   1:  PR[GP1:91,1] = PR[GP1:90,1] + -57.103;
   1:  PR[GP1:91,2] = PR[GP1:90,2] + -24.038;
   1:L PR[91] 10mm/sec CNT100;
   1:  PR[GP1:91,1] = PR[GP1:90,1] + -52.961;
   1:  PR[GP1:91,2] = PR[GP1:90,2] + -27.754;
   1:L PR[91] 10mm/sec CNT100;
   1:  PR[GP1:91,1] = PR[GP1:90,1] + -51.108;
   1:  PR[GP1:91,2] = PR[GP1:90,2] + -29.248;
   1:L PR[91] 10mm/sec CNT100;
   1:  PR[GP1:91,1] = PR[GP1:90,1] + -46.370;
   1:  PR[GP1:91,2] = PR[GP1:90,2] + -32.199;
   1:L PR[91] 10mm/sec CNT100;
   1:  PR[GP1:91,1] = PR[GP1:90,1] + -41.741;
   1:  PR[GP1:91,2] = PR[GP1:90,2] + -34.058;
   1:L PR[91] 10mm/sec CNT100;
   1:  PR[GP1:91,1] = PR[GP1:90,1] + -38.037;
   1:  PR[GP1:91,2] = PR[GP1:90,2] + -35.365;
   1:L PR[91] 10mm/sec CNT100;
   1:  PR[GP1:91,1] = PR[GP1:90,1] + -33.335;
   1:  PR[GP1:91,2] = PR[GP1:90,2] + -36.379;
   1:L PR[91] 10mm/sec CNT100;
   1:  PR[GP1:91,1] = PR[GP1:90,1] + -29.075;
   1:  PR[GP1:91,2] = PR[GP1:90,2] + -36.543;
   1:L PR[91] 10mm/sec CNT100;
   1:  PR[GP1:91,1] = PR[GP1:90,1] + -23.571;
   1:  PR[GP1:91,2] = PR[GP1:90,2] + -36.561;
   1:L PR[91] 10mm/sec CNT100;
   1:  PR[GP1:91,1] = PR[GP1:90,1] + -19.611;
   1:  PR[GP1:91,2] = PR[GP1:90,2] + -36.043;
   1:L PR[91] 10mm/sec CNT100;
   1:  PR[GP1:91,1] = PR[GP1:90,1] + -16.220;
   1:  PR[GP1:91,2] = PR[GP1:90,2] + -34.964;
   1:L PR[91] 10mm/sec CNT100;
   1:  PR[GP1:91,1] = PR[GP1:90,1] + -9.801;
   1:  PR[GP1:91,2] = PR[GP1:90,2] + -32.733;
   1:L PR[91] 10mm/sec CNT100;
   1:  PR[GP1:91,1] = PR[GP1:90,1] + -6.929;
   1:  PR[GP1:91,2] = PR[GP1:90,2] + -31.231;
   1:L PR[91] 10mm/sec CNT100;
   1:  PR[GP1:91,1] = PR[GP1:90,1] + -2.748;
   1:  PR[GP1:91,2] = PR[GP1:90,2] + -28.193;
   1:L PR[91] 10mm/sec CNT100;
   1:  PR[GP1:91,1] = PR[GP1:90,1] + 1.666;
   1:  PR[GP1:91,2] = PR[GP1:90,2] + -27.262;
   1:L PR[91] 10mm/sec CNT100;
   1:  PR[GP1:91,1] = PR[GP1:90,1] + 3.628;
   1:  PR[GP1:91,2] = PR[GP1:90,2] + -28.241;
   1:L PR[91] 10mm/sec CNT100;
   1:  PR[GP1:91,1] = PR[GP1:90,1] + 7.755;
   1:  PR[GP1:91,2] = PR[GP1:90,2] + -31.240;
   1:L PR[91] 10mm/sec CNT100;
   1:  PR[GP1:91,1] = PR[GP1:90,1] + 10.603;
   1:  PR[GP1:91,2] = PR[GP1:90,2] + -32.726;
   1:L PR[91] 10mm/sec CNT100;
   1:  PR[GP1:91,1] = PR[GP1:90,1] + 14.146;
   1:  PR[GP1:91,2] = PR[GP1:90,2] + -33.864;
   1:L PR[91] 10mm/sec CNT100;
   1:  PR[GP1:91,1] = PR[GP1:90,1] + 20.435;
   1:  PR[GP1:91,2] = PR[GP1:90,2] + -36.041;
   1:L PR[91] 10mm/sec CNT100;
   1:  PR[GP1:91,1] = PR[GP1:90,1] + 24.372;
   1:  PR[GP1:91,2] = PR[GP1:90,2] + -36.559;
   1:L PR[91] 10mm/sec CNT100;
   1:  PR[GP1:91,1] = PR[GP1:90,1] + 28.980;
   1:  PR[GP1:91,2] = PR[GP1:90,2] + -36.404;
   1:L PR[91] 10mm/sec CNT100;
   1:  PR[GP1:91,1] = PR[GP1:90,1] + 34.135;
   1:  PR[GP1:91,2] = PR[GP1:90,2] + -36.382;
   1:L PR[91] 10mm/sec CNT100;
   1:  PR[GP1:91,1] = PR[GP1:90,1] + 38.809;
   1:  PR[GP1:91,2] = PR[GP1:90,2] + -35.376;
   1:L PR[91] 10mm/sec CNT100;
   1:  PR[GP1:91,1] = PR[GP1:90,1] + 43.946;
   1:  PR[GP1:91,2] = PR[GP1:90,2] + -33.352;
   1:L PR[91] 10mm/sec CNT100;
   1:  PR[GP1:91,1] = PR[GP1:90,1] + 47.174;
   1:  PR[GP1:91,2] = PR[GP1:90,2] + -32.208;
   1:L PR[91] 10mm/sec CNT100;
   1:  PR[GP1:91,1] = PR[GP1:90,1] + 51.860;
   1:  PR[GP1:91,2] = PR[GP1:90,2] + -29.303;
   1:L PR[91] 10mm/sec CNT100;
   1:  PR[GP1:91,1] = PR[GP1:90,1] + 56.414;
   1:  PR[GP1:91,2] = PR[GP1:90,2] + -25.270;
   1:L PR[91] 10mm/sec CNT100;
   1:  PR[GP1:91,1] = PR[GP1:90,1] + 57.859;
   1:  PR[GP1:91,2] = PR[GP1:90,2] + -24.101;
   1:L PR[91] 10mm/sec CNT100;
   1:  PR[GP1:91,1] = PR[GP1:90,1] + 61.565;
   1:  PR[GP1:91,2] = PR[GP1:90,2] + -19.290;
   1:L PR[91] 10mm/sec CNT100;
   1:  PR[GP1:91,1] = PR[GP1:90,1] + 64.651;
   1:  PR[GP1:91,2] = PR[GP1:90,2] + -13.368;
   1:L PR[91] 10mm/sec CNT100;
   1:  PR[GP1:91,1] = PR[GP1:90,1] + 65.047;
   1:  PR[GP1:91,2] = PR[GP1:90,2] + -12.707;
   1:L PR[91] 10mm/sec CNT100;
   1:  PR[GP1:91,1] = PR[GP1:90,1] + 66.798;
   1:  PR[GP1:91,2] = PR[GP1:90,2] + -6.849;
   1:L PR[91] 10mm/sec CNT100;
   1:  PR[GP1:91,1] = PR[GP1:90,1] + 67.403;
   1:  PR[GP1:91,2] = PR[GP1:90,2] + -0.368;
   1:L PR[91] 10mm/sec CNT100;
   1:  PR[GP1:91,1] = PR[GP1:90,1] + 67.475;
   1:  PR[GP1:91,2] = PR[GP1:90,2] + 0.023;
   1:L PR[91] 10mm/sec CNT100;
   1:  PR[GP1:91,1] = PR[GP1:90,1] + 66.891;
   1:  PR[GP1:91,2] = PR[GP1:90,2] + 6.353;
   1:L PR[91] 10mm/sec CNT100;
   1:  PR[GP1:91,1] = PR[GP1:90,1] + 66.805;
   1:  PR[GP1:91,2] = PR[GP1:90,2] + 6.814;
   1:L PR[91] 10mm/sec CNT100;
   1:  PR[GP1:91,1] = PR[GP1:90,1] + 65.042;
   1:  PR[GP1:91,2] = PR[GP1:90,2] + 12.717;
   1:L PR[91] 10mm/sec CNT100;
   1:  PR[GP1:91,1] = PR[GP1:90,1] + 62.177;
   1:  PR[GP1:91,2] = PR[GP1:90,2] + 18.268;
   1:L PR[91] 10mm/sec CNT100;
   1:  PR[GP1:91,1] = PR[GP1:90,1] + 61.576;
   1:  PR[GP1:91,2] = PR[GP1:90,2] + 19.266;
   1:L PR[91] 10mm/sec CNT100;
   1:  PR[GP1:91,1] = PR[GP1:90,1] + 57.851;
   1:  PR[GP1:91,2] = PR[GP1:90,2] + 24.103;
   1:L PR[91] 10mm/sec CNT100;
   1:  PR[GP1:91,1] = PR[GP1:90,1] + 53.731;
   1:  PR[GP1:91,2] = PR[GP1:90,2] + 27.787;
   1:L PR[91] 10mm/sec CNT100;
   1:  PR[GP1:91,1] = PR[GP1:90,1] + 51.874;
   1:  PR[GP1:91,2] = PR[GP1:90,2] + 29.286;
   1:L PR[91] 10mm/sec CNT100;
   1:  PR[GP1:91,1] = PR[GP1:90,1] + 47.166;
   1:  PR[GP1:91,2] = PR[GP1:90,2] + 32.204;
   1:L PR[91] 10mm/sec CNT100;
   1:  PR[GP1:91,1] = PR[GP1:90,1] + 42.531;
   1:  PR[GP1:91,2] = PR[GP1:90,2] + 34.055;
   1:L PR[91] 10mm/sec CNT100;
   1:  PR[GP1:91,1] = PR[GP1:90,1] + 38.825;
   1:  PR[GP1:91,2] = PR[GP1:90,2] + 35.364;
   1:L PR[91] 10mm/sec CNT100;
   1:  PR[GP1:91,1] = PR[GP1:90,1] + 34.131;
   1:  PR[GP1:91,2] = PR[GP1:90,2] + 36.374;
   1:L PR[91] 10mm/sec CNT100;
   1:  PR[GP1:91,1] = PR[GP1:90,1] + 29.893;
   1:  PR[GP1:91,2] = PR[GP1:90,2] + 36.534;
   1:L PR[91] 10mm/sec CNT100;
   1:  PR[GP1:91,1] = PR[GP1:90,1] + 24.390;
   1:  PR[GP1:91,2] = PR[GP1:90,2] + 36.553;
   1:L PR[91] 10mm/sec CNT100;
   1:  PR[GP1:91,1] = PR[GP1:90,1] + 20.437;
   1:  PR[GP1:91,2] = PR[GP1:90,2] + 36.033;
   1:L PR[91] 10mm/sec CNT100;
   1:  PR[GP1:91,1] = PR[GP1:90,1] + 17.041;
   1:  PR[GP1:91,2] = PR[GP1:90,2] + 34.953;
   1:L PR[91] 10mm/sec CNT100;
   1:  PR[GP1:91,1] = PR[GP1:90,1] + 10.620;
   1:  PR[GP1:91,2] = PR[GP1:90,2] + 32.726;
   1:L PR[91] 10mm/sec CNT100;
   1:  PR[GP1:91,1] = PR[GP1:90,1] + 7.758;
   1:  PR[GP1:91,2] = PR[GP1:90,2] + 31.233;
   1:L PR[91] 10mm/sec CNT100;
   1:  PR[GP1:91,1] = PR[GP1:90,1] + 4.694;
   1:  PR[GP1:91,2] = PR[GP1:90,2] + 29.068;
   1:L PR[91] 10mm/sec CNT100;
   1:  PR[GP1:91,1] = PR[GP1:90,1] + 4.167;
   1:  PR[GP1:91,2] = PR[GP1:90,2] + 28.656;
   1:L PR[91] 10mm/sec CNT100;
   1:  PR[GP1:91,1] = PR[GP1:90,1] + 3.676;
   1:  PR[GP1:91,2] = PR[GP1:90,2] + 28.085;
   1:L PR[91] 10mm/sec CNT100;
   1:  PR[GP1:91,1] = PR[GP1:90,1] + 1.967;
   1:  PR[GP1:91,2] = PR[GP1:90,2] + 27.410;
   1:L PR[91] 10mm/sec CNT100;
   1:  PR[GP1:91,1] = PR[GP1:90,1] + 1.682;
   1:  PR[GP1:91,2] = PR[GP1:90,2] + 27.251;
   1:L PR[91] 10mm/sec CNT100;
   1:  PR[GP1:91,1] = PR[GP1:90,1] + 1.109;
   1:  PR[GP1:91,2] = PR[GP1:90,2] + 27.857;
   1:  PR[GP1:91,3] = PR[GP1:90,3] + 57.190;
   1:L PR[91] 10mm/sec CNT100;
   1:  PR[GP1:91,1] = PR[GP1:90,1] + -1.208;
   1:  PR[GP1:91,2] = PR[GP1:90,2] + 28.395;
   1:L PR[91] 10mm/sec CNT100;
   1:  PR[GP1:91,1] = PR[GP1:90,1] + -2.475;
   1:  PR[GP1:91,2] = PR[GP1:90,2] + 28.558;
   1:L PR[91] 10mm/sec CNT100;
   1:  PR[GP1:91,1] = PR[GP1:90,1] + -2.815;
   1:  PR[GP1:91,2] = PR[GP1:90,2] + 28.731;
   1:L PR[91] 10mm/sec CNT100;
   1:  PR[GP1:91,1] = PR[GP1:90,1] + -3.006;
   1:  PR[GP1:91,2] = PR[GP1:90,2] + 28.953;
   1:L PR[91] 10mm/sec CNT100;
   1:  PR[GP1:91,1] = PR[GP1:90,1] + -3.157;
   1:  PR[GP1:91,2] = PR[GP1:90,2] + 29.072;
   1:L PR[91] 10mm/sec CNT100;
   1:  PR[GP1:91,1] = PR[GP1:90,1] + -6.473;
   1:  PR[GP1:91,2] = PR[GP1:90,2] + 31.415;
   1:L PR[91] 10mm/sec CNT100;
   1:  PR[GP1:91,1] = PR[GP1:90,1] + -9.060;
   1:  PR[GP1:91,2] = PR[GP1:90,2] + 32.768;
   1:L PR[91] 10mm/sec CNT100;
   1:  PR[GP1:91,1] = PR[GP1:90,1] + -12.256;
   1:  PR[GP1:91,2] = PR[GP1:90,2] + 33.795;
   1:L PR[91] 10mm/sec CNT100;
   1:  PR[GP1:91,1] = PR[GP1:90,1] + -19.196;
   1:  PR[GP1:91,2] = PR[GP1:90,2] + 36.194;
   1:L PR[91] 10mm/sec CNT100;
   1:  PR[GP1:91,1] = PR[GP1:90,1] + -22.805;
   1:  PR[GP1:91,2] = PR[GP1:90,2] + 36.666;
   1:L PR[91] 10mm/sec CNT100;
   1:  PR[GP1:91,1] = PR[GP1:90,1] + -27.050;
   1:  PR[GP1:91,2] = PR[GP1:90,2] + 36.520;
   1:L PR[91] 10mm/sec CNT100;
   1:  PR[GP1:91,1] = PR[GP1:90,1] + -32.941;
   1:  PR[GP1:91,2] = PR[GP1:90,2] + 36.491;
   1:L PR[91] 10mm/sec CNT100;
   1:  PR[GP1:91,1] = PR[GP1:90,1] + -37.277;
   1:  PR[GP1:91,2] = PR[GP1:90,2] + 35.555;
   1:L PR[91] 10mm/sec CNT100;
   1:  PR[GP1:91,1] = PR[GP1:90,1] + -42.036;
   1:  PR[GP1:91,2] = PR[GP1:90,2] + 33.671;
   1:L PR[91] 10mm/sec CNT100;
   1:  PR[GP1:91,1] = PR[GP1:90,1] + -45.983;
   1:  PR[GP1:91,2] = PR[GP1:90,2] + 32.269;
   1:L PR[91] 10mm/sec CNT100;
   1:  PR[GP1:91,1] = PR[GP1:90,1] + -50.389;
   1:  PR[GP1:91,2] = PR[GP1:90,2] + 29.524;
   1:L PR[91] 10mm/sec CNT100;
   1:  PR[GP1:91,1] = PR[GP1:90,1] + -54.674;
   1:  PR[GP1:91,2] = PR[GP1:90,2] + 25.720;
   1:L PR[91] 10mm/sec CNT100;
   1:  PR[GP1:91,1] = PR[GP1:90,1] + -56.714;
   1:  PR[GP1:91,2] = PR[GP1:90,2] + 24.069;
   1:L PR[91] 10mm/sec CNT100;
   1:  PR[GP1:91,1] = PR[GP1:90,1] + -60.161;
   1:  PR[GP1:91,2] = PR[GP1:90,2] + 19.583;
   1:L PR[91] 10mm/sec CNT100;
   1:  PR[GP1:91,1] = PR[GP1:90,1] + -63.055;
   1:  PR[GP1:91,2] = PR[GP1:90,2] + 13.966;
   1:L PR[91] 10mm/sec CNT100;
   1:  PR[GP1:91,1] = PR[GP1:90,1] + -63.845;
   1:  PR[GP1:91,2] = PR[GP1:90,2] + 12.647;
   1:L PR[91] 10mm/sec CNT100;
   1:  PR[GP1:91,1] = PR[GP1:90,1] + -65.497;
   1:  PR[GP1:91,2] = PR[GP1:90,2] + 7.041;
   1:L PR[91] 10mm/sec CNT100;
   1:  PR[GP1:91,1] = PR[GP1:90,1] + -66.042;
   1:  PR[GP1:91,2] = PR[GP1:90,2] + 1.088;
   1:L PR[91] 10mm/sec CNT100;
   1:  PR[GP1:91,1] = PR[GP1:90,1] + -66.248;
   1:  PR[GP1:91,2] = PR[GP1:90,2] + -0.032;
   1:L PR[91] 10mm/sec CNT100;
   1:  PR[GP1:91,1] = PR[GP1:90,1] + -65.723;
   1:  PR[GP1:91,2] = PR[GP1:90,2] + -5.850;
   1:L PR[91] 10mm/sec CNT100;
   1:  PR[GP1:91,1] = PR[GP1:90,1] + -65.505;
   1:  PR[GP1:91,2] = PR[GP1:90,2] + -7.023;
   1:L PR[91] 10mm/sec CNT100;
   1:  PR[GP1:91,1] = PR[GP1:90,1] + -63.839;
   1:  PR[GP1:91,2] = PR[GP1:90,2] + -12.676;
   1:L PR[91] 10mm/sec CNT100;
   1:  PR[GP1:91,1] = PR[GP1:90,1] + -61.145;
   1:  PR[GP1:91,2] = PR[GP1:90,2] + -17.958;
   1:L PR[91] 10mm/sec CNT100;
   1:  PR[GP1:91,1] = PR[GP1:90,1] + -60.172;
   1:  PR[GP1:91,2] = PR[GP1:90,2] + -19.577;
   1:L PR[91] 10mm/sec CNT100;
   1:  PR[GP1:91,1] = PR[GP1:90,1] + -56.703;
   1:  PR[GP1:91,2] = PR[GP1:90,2] + -24.092;
   1:L PR[91] 10mm/sec CNT100;
   1:  PR[GP1:91,1] = PR[GP1:90,1] + -52.808;
   1:  PR[GP1:91,2] = PR[GP1:90,2] + -27.585;
   1:L PR[91] 10mm/sec CNT100;
   1:  PR[GP1:91,1] = PR[GP1:90,1] + -50.399;
   1:  PR[GP1:91,2] = PR[GP1:90,2] + -29.527;
   1:L PR[91] 10mm/sec CNT100;
   1:  PR[GP1:91,1] = PR[GP1:90,1] + -45.969;
   1:  PR[GP1:91,2] = PR[GP1:90,2] + -32.287;
   1:L PR[91] 10mm/sec CNT100;
   1:  PR[GP1:91,1] = PR[GP1:90,1] + -41.641;
   1:  PR[GP1:91,2] = PR[GP1:90,2] + -34.025;
   1:L PR[91] 10mm/sec CNT100;
   1:  PR[GP1:91,1] = PR[GP1:90,1] + -37.282;
   1:  PR[GP1:91,2] = PR[GP1:90,2] + -35.563;
   1:L PR[91] 10mm/sec CNT100;
   1:  PR[GP1:91,1] = PR[GP1:90,1] + -32.924;
   1:  PR[GP1:91,2] = PR[GP1:90,2] + -36.503;
   1:L PR[91] 10mm/sec CNT100;
   1:  PR[GP1:91,1] = PR[GP1:90,1] + -28.976;
   1:  PR[GP1:91,2] = PR[GP1:90,2] + -36.655;
   1:L PR[91] 10mm/sec CNT100;
   1:  PR[GP1:91,1] = PR[GP1:90,1] + -22.803;
   1:  PR[GP1:91,2] = PR[GP1:90,2] + -36.674;
   1:L PR[91] 10mm/sec CNT100;
   1:  PR[GP1:91,1] = PR[GP1:90,1] + -19.178;
   1:  PR[GP1:91,2] = PR[GP1:90,2] + -36.201;
   1:L PR[91] 10mm/sec CNT100;
   1:  PR[GP1:91,1] = PR[GP1:90,1] + -16.071;
   1:  PR[GP1:91,2] = PR[GP1:90,2] + -35.212;
   1:L PR[91] 10mm/sec CNT100;
   1:  PR[GP1:91,1] = PR[GP1:90,1] + -9.055;
   1:  PR[GP1:91,2] = PR[GP1:90,2] + -32.774;
   1:L PR[91] 10mm/sec CNT100;
   1:  PR[GP1:91,1] = PR[GP1:90,1] + -6.469;
   1:  PR[GP1:91,2] = PR[GP1:90,2] + -31.421;
   1:L PR[91] 10mm/sec CNT100;
   1:  PR[GP1:91,1] = PR[GP1:90,1] + -2.643;
   1:  PR[GP1:91,2] = PR[GP1:90,2] + -28.641;
   1:L PR[91] 10mm/sec CNT100;
   1:  PR[GP1:91,1] = PR[GP1:90,1] + -2.154;
   1:  PR[GP1:91,2] = PR[GP1:90,2] + -28.622;
   1:L PR[91] 10mm/sec CNT100;
   1:  PR[GP1:91,1] = PR[GP1:90,1] + 1.805;
   1:  PR[GP1:91,2] = PR[GP1:90,2] + -27.777;
   1:L PR[91] 10mm/sec CNT100;
   1:  PR[GP1:91,1] = PR[GP1:90,1] + 2.022;
   1:  PR[GP1:91,2] = PR[GP1:90,2] + -27.952;
   1:L PR[91] 10mm/sec CNT100;
   1:  PR[GP1:91,1] = PR[GP1:90,1] + 3.566;
   1:  PR[GP1:91,2] = PR[GP1:90,2] + -28.721;
   1:L PR[91] 10mm/sec CNT100;
   1:  PR[GP1:91,1] = PR[GP1:90,1] + 7.294;
   1:  PR[GP1:91,2] = PR[GP1:90,2] + -31.429;
   1:L PR[91] 10mm/sec CNT100;
   1:  PR[GP1:91,1] = PR[GP1:90,1] + 9.857;
   1:  PR[GP1:91,2] = PR[GP1:90,2] + -32.767;
   1:L PR[91] 10mm/sec CNT100;
   1:  PR[GP1:91,1] = PR[GP1:90,1] + 13.052;
   1:  PR[GP1:91,2] = PR[GP1:90,2] + -33.793;
   1:L PR[91] 10mm/sec CNT100;
   1:  PR[GP1:91,1] = PR[GP1:90,1] + 20.002;
   1:  PR[GP1:91,2] = PR[GP1:90,2] + -36.199;
   1:L PR[91] 10mm/sec CNT100;
   1:  PR[GP1:91,1] = PR[GP1:90,1] + 23.605;
   1:  PR[GP1:91,2] = PR[GP1:90,2] + -36.673;
   1:L PR[91] 10mm/sec CNT100;
   1:  PR[GP1:91,1] = PR[GP1:90,1] + 27.830;
   1:  PR[GP1:91,2] = PR[GP1:90,2] + -36.531;
   1:L PR[91] 10mm/sec CNT100;
   1:  PR[GP1:91,1] = PR[GP1:90,1] + 33.727;
   1:  PR[GP1:91,2] = PR[GP1:90,2] + -36.505;
   1:L PR[91] 10mm/sec CNT100;
